	pH_4_END:
		IF timerDoCalibration.Q THEN
			timerDoCalibration.IN := FALSE;
			bBusy := FALSE;
			eSMState := WAIT;
		END_IF
	
	
	pH_10_START:
		nCalOutputPH10 := TRUE;
		timerBtnPress.IN := TRUE;
		IF timerBtnPress.Q THEN
			nCalOutputPH10 := FALSE;
			eSMState := pH_10_END;
			timerBtnPress.IN := FALSE; 
			timerDoCalibration.IN := TRUE;
		END_IF
		
		eSMState := pH_10_END;
			
			
		
	pH_10_END:
		IF timerDoCalibration.Q THEN
			timerDoCalibration.IN := FALSE;
			bBusy := FALSE;
			eSMState := WAIT;
		END_IF

END_CASE

METHOD PRIVATE calculate : BOOL
VAR_INPUT
	
	// Var
END_VAR
VAR
	nMeasuredCurrent: REAL;
END_VAR
nMeasuredCurrent := (INT_TO_REAL(nRawInput)/GVL.nMaxADCOutput)*16.0 + 4.0; // in mA

// nCurrentValue := (nMeasuredCurrent - 4.0) * (14.0 / 16.0);  // equation is PH = (mA reading - 4.0) * (14.0 / 16.0)
nCurrentValue := (nMeasuredCurrent - 4.0) * (14.0 / 16.0);  // equation is PH = (mA reading - 4.0) * (14.0 / 16.0)
END_METHOD

METHOD calibrate : BOOL
VAR_INPUT
	PhUnderTest: INT; // Can be 4, 7, or 10 (7 must be done first if doing multiple)
END_VAR
CASE PhUnderTest OF
	4:
		eSMState := pH_4_START;
	7:
		eSMState := pH_7_START;
	10:
		eSMState := pH_10_START;
END_CASE

bBusy := TRUE;
END_METHOD

{warning 'add method implementation '}
METHOD disable : BOOL
bEnable := FALSE;
END_METHOD

{warning 'add method implementation '}
METHOD enable : BOOL
bEnable := TRUE;
END_METHOD

{warning 'add method implementation '}
METHOD FB_init : BOOL
VAR_INPUT
	(* if TRUE, the retain variables are initialized (warm start / cold start)*)
	bInitRetains	: BOOL;
	(* if TRUE, the instance afterwards gets moved into the copy code (online change)*)
	bInCopyCode	: BOOL;
	
	SensorID	: STRING(80);
	SensorDescr	: STRING(255);
	SensorType	: E_SensorType;
END_VAR
sID := SensorID;
sDescr := SensorDescr;
eSensorType := SensorType;
END_METHOD

{warning 'add method implementation '}
METHOD getType : E_SensorType
getType := eSensorType;
END_METHOD

{warning 'add method implementation '}
METHOD getValue : REAL
getValue := nCurrentValue;
END_METHOD

{warning 'add method implementation '}
METHOD write : BOOL
// use this method to initiated a hardware read from assigned IO if required
END_METHOD

END_FUNCTION_BLOCK

// ---- POUs/02 Sensors/Dosing Machine/FB_Sensor_AtlasTEMP.TcPOU
{attribute 'OPC.UA.DA.StructuredType' := '1'}
FUNCTION_BLOCK FB_Sensor_AtlasTEMP EXTENDS FB_BaseDevice IMPLEMENTS I_Device, I_Sensor


VAR
	{attribute 'OPC.UA.DA' := '0'} 
	eSensorType: E_SensorType;
	{attribute 'OPC.UA.DA' := '0'} 
	nRawInput AT %I*: INT;
	nFaultInput AT %I*: BOOL;
	{attribute 'OPC.UA.DA' := '1'} 
	nCurrentValue: REAL;
	
	{attribute 'OPC.UA.DA' := '0'} 
	nCalOutput1 AT %Q*: BOOL;
	{attribute 'OPC.UA.DA' := '0'} 
	nCalOutput2 AT %Q*: BOOL;
	{attribute 'OPC.UA.DA' := '0'} 
	nCalOutput3 AT %Q*: BOOL;
	
	{attribute 'OPC.UA.DA' := '0'} 
	trigCalibrate: R_TRIG;
	{attribute 'OPC.UA.DA' := '0'} 
	timerBtnPress: TON := (PT:=T#250MS,IN := FALSE);
	
	{attribute 'OPC.UA.DA' := '0'} 
	timerDoCalibration: TON := (PT:=T#120S,IN := FALSE); // Check this time during testing! The instructions are not clear about what happens after initiating a calibration request 
	
	{attribute 'OPC.UA.DA' := '0'} 
	eSMState: (WAIT, CAL_START, CAL_FINISH) := WAIT;
	
END_VAR

calculate();

CASE eSMState OF 
	WAIT:
		// wait for the calibrate method call to change the ESMState variable
		
	CAL_START:
		nCalOutput1 := TRUE;
		timerBtnPress.IN := TRUE;
		IF timerBtnPress.Q THEN
			nCalOutput1 := FALSE;
			eSMState := CAL_FINISH;
			timerBtnPress.IN := FALSE; 
			timerDoCalibration.IN := TRUE;
		END_IF
		
		eSMState := CAL_FINISH;
		
	CAL_FINISH:
		IF timerDoCalibration.Q THEN
			timerDoCalibration.IN := FALSE;			// CHeck the functionality of this step - instructions are not clear
			bBusy := FALSE;
			eSMState := WAIT;
		END_IF
		
END_CASE

METHOD PRIVATE calculate : BOOL
VAR_INPUT
	
	// Var
END_VAR

VAR
	nMeasuredCurrent: REAL;
END_VAR
nMeasuredCurrent := (INT_TO_REAL(nRawInput)/GVL.nMaxADCOutput)*16.0 + 4.0; // in mA


nCurrentValue := (((nMeasuredCurrent - 4.0) / 16.0) * 360.0)- 180;  // equation is TEMP =    [(mA reading - 4.0)* 275 / 16 ] - 55

// nCurrentValue := (((nMeasuredCurrent - 4.0) * 275.0 / 16.0))- 55;  // equation is TEMP =    [(mA reading - 4.0)* 275 / 16 ] - 55

// This equation is for the default probe type 'Option 1' with a range of -55 to 220 deg C
END_METHOD

METHOD calibrate : BOOL
VAR_INPUT
END_VAR
// The user manual only shows a manual calibration method
// Perhaps this probe does not need to be calibrated as often and the PLC method is not offered? Need to investigate

eSMState := CAL_START;
END_METHOD

{warning 'add method implementation '}
METHOD disable : BOOL
bEnable := FALSE;
END_METHOD

{warning 'add method implementation '}
METHOD enable : BOOL
bEnable := TRUE;
END_METHOD

{warning 'add method implementation '}
METHOD FB_init : BOOL
VAR_INPUT
	(* if TRUE, the retain variables are initialized (warm start / cold start)*)
	bInitRetains	: BOOL;
	(* if TRUE, the instance afterwards gets moved into the copy code (online change)*)
	bInCopyCode	: BOOL;
	
	SensorID	: STRING(80);
	SensorDescr	: STRING(255);
	SensorType	: E_SensorType;
END_VAR
sID := SensorID;
sDescr := SensorDescr;
eSensorType := SensorType;
END_METHOD

{warning 'add method implementation '}
METHOD getType : E_SensorType
getType := eSensorType;
END_METHOD

{warning 'add method implementation '}
METHOD getValue : REAL
getValue := nCurrentValue;
END_METHOD

{warning 'add method implementation '}
METHOD write : BOOL
// use this method to initiated a hardware read from assigned IO if required
END_METHOD

END_FUNCTION_BLOCK

// ---- POUs/02 Sensors/Dosing Machine/FB_Sensor_GrowMedium_EC.TcPOU
{attribute 'OPC.UA.DA.StructuredType' := '1'}
FUNCTION_BLOCK FB_Sensor_GrowMedium_EC EXTENDS FB_BaseSensor IMPLEMENTS I_Device, I_Sensor

VAR
	
	bCAL: BOOL := FALSE;
	
	eSMState: (WAIT, CAL_LOW, CAL_HIGH, CALC_CORRECTION) := WAIT;

END_VAR
	
VAR PERSISTENT ;
	nECLOW_val: REAL;
	nECHIGH_val: REAL;
	
	nCurveGradient: REAL := 0.625; // 
	nCurveOffset: REAL := -2.5; // Defaults
END_VAR

calculate();
filter();

// Detect if any buttons in ignition have been pressed for Calibration
IF bCAL THEN 
	bCAL := FALSE;
	CASE eSMState OF
		WAIT:
			eSMState := CAL_LOW;
		CAL_LOW:
			eSMState := CAL_HIGH;
		CAL_HIGH:
			eSMState := CALC_CORRECTION;
	END_CASE
END_IF


CASE eSMState OF 
	WAIT:
		// wait here for a calibration command to be received
		eState := E_DeviceState.RUNNING;


	CAL_LOW:
		nECLOW_val := nMeasuredCurrent;
		eState := E_DeviceState.CAL_STEP1;

	CAL_HIGH:
		nECHIGH_val := nMeasuredCurrent;
		eState := E_DeviceState.CAL_STEP2;
	
	CALC_CORRECTION:
		nCurveGradient := ((1413.0-84.0)/1000.0) / (nECHIGH_val - nECLOW_val);
		nCurveOffset := (84.0/1000.0) - (nCurveGradient * nECLOW_val);
		eSMState := WAIT;
		eState := E_DeviceState.CAL_STEP3;
		
		
END_CASE

METHOD PRIVATE calculate : BOOL
VAR_INPUT
	
END_VAR
nMeasuredCurrent := (INT_TO_REAL(nRawInput)/GVL.nMaxADCOutput)*16.0 + 4.0; // in mA

// nCurrentValue := (nCurveGradient * nMeasuredCurrent) + nCurveOffset;

nCurrentValue := (nCurveGradient * nFilteredCurrent) + nCurveOffset; // delete this eventually
END_METHOD

METHOD calibrate : BOOL
VAR_INPUT
	
END_VAR
bCAL := TRUE;
END_METHOD

{warning 'add method implementation '}
METHOD disable : BOOL
bEnable := FALSE;
END_METHOD

{warning 'add method implementation '}
METHOD enable : BOOL
bEnable := TRUE;
END_METHOD

{warning 'add method implementation '}
METHOD FB_init : BOOL
VAR_INPUT
	(* if TRUE, the retain variables are initialized (warm start / cold start)*)
	bInitRetains	: BOOL;
	(* if TRUE, the instance afterwards gets moved into the copy code (online change)*)
	bInCopyCode	: BOOL;
	
	SensorID	: STRING(80);
	SensorDescr	: STRING(255);
	SensorType	: E_SensorType;
END_VAR
sID := SensorID;
sDescr := SensorDescr;
eSensorType := SensorType;
END_METHOD

{warning 'add method implementation '}
METHOD getType : E_SensorType
getType := eSensorType;
END_METHOD

{warning 'add method implementation '}
METHOD getValue : REAL
getValue := nCurrentValue;
END_METHOD

{warning 'add method implementation '}
METHOD write : BOOL
// use this method to initiated a hardware read from assigned IO if required
END_METHOD

END_FUNCTION_BLOCK

// ---- POUs/02 Sensors/Dosing Machine/FB_Sensor_GrowMedium_MOISTURE.TcPOU
{attribute 'OPC.UA.DA.StructuredType' := '1'}
FUNCTION_BLOCK FB_Sensor_GrowMedium_MOISTURE EXTENDS FB_BaseSensor IMPLEMENTS I_Device, I_Sensor

VAR
	
	bCAL: BOOL := FALSE;
	
	eSMState: (WAIT, CAL_DRY, CAL_WET, CALC_CORRECTION) := WAIT;

END_VAR
	
VAR PERSISTENT ;
	nMoisture_LOW_val: REAL;
	nMoisture_HIGH_val: REAL;
	
	nCurveGradient: REAL := 0.625; // 
	nCurveOffset: REAL := -2.5; // Defaults
END_VAR

calculate();
filter();

// Detect if any buttons in ignition have been pressed for Calibration
IF bCAL THEN 
	bCAL := FALSE;
	CASE eSMState OF
		WAIT:
			eSMState := CAL_DRY;
		CAL_DRY:
			eSMState := CAL_WET;
		CAL_WET:
			eSMState := CALC_CORRECTION;
	END_CASE
END_IF


CASE eSMState OF 
	WAIT:
		// wait here for a calibration command to be received
		eState := E_DeviceState.RUNNING;
	CAL_DRY:
		nMoisture_LOW_val 	:= nMeasuredCurrent;
		eState := E_DeviceState.CAL_STEP1;

	CAL_WET:
		nMoisture_HIGH_val 	:= nMeasuredCurrent;
		eState := E_DeviceState.CAL_STEP2;

	CALC_CORRECTION:
		nCurveGradient := 100.0 / (nMoisture_HIGH_val - nMoisture_LOW_val);
		nCurveOffset := 100.0 - (nCurveGradient * nMoisture_HIGH_val);
		eState := E_DeviceState.CAL_STEP3;
		eSMState := WAIT;
		
END_CASE

METHOD PRIVATE calculate : BOOL
VAR_INPUT
	
END_VAR
nMeasuredCurrent := (INT_TO_REAL(nRawInput)/GVL.nMaxADCOutput)*16.0 + 4.0; // in mA

// nCurrentValue := (nCurveGradient * nMeasuredCurrent) + nCurveOffset;

nCurrentValue := (nCurveGradient * nFilteredCurrent) + nCurveOffset; // delete this eventually
END_METHOD

METHOD calibrate : BOOL
VAR_INPUT
	
END_VAR

bCAL := TRUE;
END_METHOD

{warning 'add method implementation '}
METHOD disable : BOOL
bEnable := FALSE;
END_METHOD

{warning 'add method implementation '}
METHOD enable : BOOL
bEnable := TRUE;
END_METHOD

{warning 'add method implementation '}
METHOD FB_init : BOOL
VAR_INPUT
	(* if TRUE, the retain variables are initialized (warm start / cold start)*)
	bInitRetains	: BOOL;
	(* if TRUE, the instance afterwards gets moved into the copy code (online change)*)
	bInCopyCode	: BOOL;
	
	SensorID	: STRING(80);
	SensorDescr	: STRING(255);
	SensorType	: E_SensorType;
END_VAR
sID := SensorID;
sDescr := SensorDescr;
eSensorType := SensorType;
END_METHOD

{warning 'add method implementation '}
METHOD getType : E_SensorType
getType := eSensorType;
END_METHOD

{warning 'add method implementation '}
METHOD getValue : REAL
getValue := nCurrentValue;
END_METHOD

{warning 'add method implementation '}
METHOD write : BOOL
// use this method to initiated a hardware read from assigned IO if required
END_METHOD

END_FUNCTION_BLOCK

// ---- POUs/02 Sensors/Dosing Machine/FB_Sensor_GrowMedium_PH.TcPOU
{attribute 'OPC.UA.DA.StructuredType' := '1'}
FUNCTION_BLOCK FB_Sensor_GrowMedium_PH EXTENDS FB_BaseSensor IMPLEMENTS I_Device, I_Sensor

VAR

	bCAL: BOOL := FALSE;
	eSMState: (WAIT, CAL_4, CAL_7, CALC_CORRECTION) := WAIT;
	
END_VAR
	
VAR PERSISTENT 

	nPH4_val: REAL;
	nPH7_val: REAL;
	
	b4High_0_20High_1: BOOL := TRUE;
	
	nCurveGradient: REAL := 6.0/16.0; // Sensor range is PH 3 to 9 over 16mA range (4-20mA)
	nCurveOffset: REAL := 1.5; 
END_VAR

calculate();
filter();

// Detect if any buttons in ignition have been pressed for Calibration
IF bCAL THEN 
	bCAL := FALSE;
	CASE eSMState OF
		WAIT:
			eSMState := CAL_4;
		CAL_4:
			eSMState := CAL_7;
		CAL_7:
			eSMState := CALC_CORRECTION;
	END_CASE
END_IF




CASE eSMState OF 
	WAIT:
		// wait here for a calibration command to be received
		eState := E_DeviceState.RUNNING;
		
	CAL_4:
		nPH4_val := nFilteredCurrent;
		eState := E_DeviceState.CAL_STEP1;

	CAL_7:
		nPH7_val := nFilteredCurrent;
		eState := E_DeviceState.CAL_STEP2;

	CALC_CORRECTION:
		nCurveGradient := 3.0 / (nPH7_val - nPH4_val);
		nCurveOffset := 4.0 - (nCurveGradient * nPH4_val);
		eState := E_DeviceState.CAL_STEP3;
		eSMState := WAIT;
		
END_CASE

METHOD PRIVATE calculate : BOOL
VAR_INPUT
	
END_VAR
IF b4High_0_20High_1 THEN
	nMeasuredCurrent := (INT_TO_REAL(nRawInput)/GVL.nMaxADCOutput)*16.0 + 4.0; // in mA
ELSE
	nMeasuredCurrent := 20.0 - (INT_TO_REAL(nRawInput)/GVL.nMaxADCOutput)*16.00; 
END_IF


// nCurrentValue := (nCurveGradient * nMeasuredCurrent) + nCurveOffset; 

nCurrentValue := (nCurveGradient * nFilteredCurrent) + nCurveOffset; // delete this eventually

nCurrentValueFiltered := (nCurveGradient * nFilteredCurrent) + nCurveOffset;
END_METHOD

METHOD calibrate : BOOL
VAR_INPUT
	
END_VAR

bCAL := TRUE;
END_METHOD

{warning 'add method implementation '}
METHOD disable : BOOL
bEnable := FALSE;
END_METHOD

{warning 'add method implementation '}
METHOD enable : BOOL
bEnable := TRUE;
END_METHOD

{warning 'add method implementation '}
METHOD FB_init : BOOL
VAR_INPUT
	(* if TRUE, the retain variables are initialized (warm start / cold start)*)
	bInitRetains	: BOOL;
	(* if TRUE, the instance afterwards gets moved into the copy code (online change)*)
	bInCopyCode	: BOOL;
	
	SensorID	: STRING(80);
	SensorDescr	: STRING(255);
	SensorType	: E_SensorType;
END_VAR
sID := SensorID;
sDescr := SensorDescr;
eSensorType := SensorType;
END_METHOD

{warning 'add method implementation '}
METHOD getType : E_SensorType
getType := eSensorType;
END_METHOD

{warning 'add method implementation '}
METHOD getValue : REAL
getValue := nCurrentValue;
END_METHOD

{warning 'add method implementation '}
METHOD write : BOOL
// use this method to initiated a hardware read from assigned IO if required
END_METHOD

END_FUNCTION_BLOCK

// ---- POUs/02 Sensors/Dosing Machine/FB_Sensor_IFM_PG2453.TcPOU
{attribute 'OPC.UA.DA.StructuredType' := '1'}
FUNCTION_BLOCK FB_Sensor_IFM_PG2453 EXTENDS FB_BaseDevice IMPLEMENTS I_Device, I_Sensor

VAR

	{attribute 'OPC.UA.DA' := '0'} 
	eSensorType: E_SensorType;
	{attribute 'OPC.UA.DA' := '0'} 
	nRawInput AT %I*: INT;
	{attribute 'OPC.UA.DA' := '1'} 
	nCurrentValue: REAL;
	
	{attribute 'OPC.UA.DA' := '1'} 
	nVal4mA: REAL;
	{attribute 'OPC.UA.DA' := '1'} 
	nVal20mA: REAL;
END_VAR

calculate();

METHOD calculate : BOOL
VAR_INPUT
END_VAR
nCurrentValue := nVal4mA + (INT_TO_REAL(nRawInput) / GVL.nMaxADCOutput) * (nVal20mA - nVal4mA) ;
END_METHOD

{warning 'add method implementation '}
METHOD disable : BOOL
bEnable := FALSE;
END_METHOD

{warning 'add method implementation '}
METHOD enable : BOOL
bEnable := TRUE;
END_METHOD

{warning 'add method implementation '}
METHOD FB_init : BOOL
VAR_INPUT
	(* if TRUE, the retain variables are initialized (warm start / cold start)*)
	bInitRetains	: BOOL;
	(* if TRUE, the instance afterwards gets moved into the copy code (online change)*)
	bInCopyCode	: BOOL;
	SensorID	: STRING(80);
	SensorDescr	: STRING(255);
	SensorType	: E_SensorType;
	
END_VAR
sID := SensorID;
sDescr := SensorDescr;
eSensorType := SensorType;
END_METHOD

{warning 'add method implementation '}
METHOD getType : E_SensorType
getType := eSensorType;
END_METHOD

{warning 'add method implementation '}
METHOD getValue : REAL
getValue := nCurrentValue;
END_METHOD

METHOD setLimits : BOOL
VAR_INPUT
	Val_4mA: 	REAL;
	Val_20mA: 	REAL;
END_VAR
nVal4mA := Val_4mA;
nVal20mA := Val_20mA;
END_METHOD

{warning 'add method implementation '}
METHOD write : BOOL
END_METHOD

END_FUNCTION_BLOCK

// ---- POUs/02 Sensors/Dosing Machine/FB_Sensor_OceanControlsPressureTx_BVS006NA.TcPOU
{attribute 'OPC.UA.DA.StructuredType' := '1'}
FUNCTION_BLOCK FB_Sensor_OceanControlsPressureTx_BVS006NA EXTENDS FB_BaseDevice IMPLEMENTS I_Device, I_Sensor
// This is a 0 to 6BAR pressure sensor from 4mA to 20mA

VAR

	{attribute 'OPC.UA.DA' := '0'} 
	eSensorType: E_SensorType;
	{attribute 'OPC.UA.DA' := '0'} 
	nRawInput AT %I*: INT;
	{attribute 'OPC.UA.DA' := '1'} 
	nCurrentValue: REAL;
	
	{attribute 'OPC.UA.DA' := '1'} 
	nVal4mA: REAL := 0; //kPA
	{attribute 'OPC.UA.DA' := '1'} 
	nVal20mA: REAL := 600; //kPA
	
END_VAR

calculate();

METHOD calculate : BOOL
VAR_INPUT
END_VAR
nCurrentValue := nVal4mA + (INT_TO_REAL(nRawInput) / GVL.nMaxADCOutput) * (nVal20mA - nVal4mA) ;
END_METHOD

{warning 'add method implementation '}
METHOD disable : BOOL
bEnable := FALSE;
END_METHOD

{warning 'add method implementation '}
METHOD enable : BOOL
bEnable := TRUE;
END_METHOD

{warning 'add method implementation '}
METHOD FB_init : BOOL
VAR_INPUT
	(* if TRUE, the retain variables are initialized (warm start / cold start)*)
	bInitRetains	: BOOL;
	(* if TRUE, the instance afterwards gets moved into the copy code (online change)*)
	bInCopyCode	: BOOL;
	SensorID	: STRING(80);
	SensorDescr	: STRING(255);
	SensorType	: E_SensorType;
	
END_VAR
sID := SensorID;
sDescr := SensorDescr;
eSensorType := SensorType;
END_METHOD

{warning 'add method implementation '}
METHOD getType : E_SensorType
getType := eSensorType;
END_METHOD

{warning 'add method implementation '}
METHOD getValue : REAL
getValue := nCurrentValue;
END_METHOD

METHOD setLimits : BOOL
VAR_INPUT
	Val_4mA: 	REAL;
	Val_20mA: 	REAL;
END_VAR
nVal4mA := Val_4mA;
nVal20mA := Val_20mA;
END_METHOD

{warning 'add method implementation '}
METHOD write : BOOL
END_METHOD

END_FUNCTION_BLOCK

// ---- POUs/02 Sensors/Dosing Machine/FB_Sensor_SICKLevelSwitch_GRF18S.TcPOU
{attribute 'OPC.UA.DA.StructuredType' := '1'}
FUNCTION_BLOCK FB_Sensor_SICKLevelSwitch_GRF18S EXTENDS FB_BaseDevice IMPLEMENTS I_Device, I_Sensor

VAR
	
	{attribute 'OPC.UA.DA' := '0'} 
	eSensorType: E_SensorType;
	{attribute 'OPC.UA.DA' := '0'} 
	nRawInput AT %I*: BOOL;
	{attribute 'OPC.UA.DA' := '1'} 
	nCurrentValue: REAL;
END_VAR

calculate();

METHOD calculate : BOOL
VAR_INPUT
END_VAR
IF nRawInput THEN
	nCurrentValue := 1;
ELSE
	nCurrentValue := 0;
END_IF
END_METHOD

{warning 'add method implementation '}
METHOD disable : BOOL
bEnable := FALSE;
END_METHOD

{warning 'add method implementation '}
METHOD enable : BOOL
bEnable := TRUE;
END_METHOD

{warning 'add method implementation '}
METHOD FB_init : BOOL
VAR_INPUT
	(* if TRUE, the retain variables are initialized (warm start / cold start)*)
	bInitRetains	: BOOL;
	(* if TRUE, the instance afterwards gets moved into the copy code (online change)*)
	bInCopyCode	: BOOL;
	SensorID	: STRING(80);
	SensorDescr	: STRING(255);
	SensorType	: E_SensorType;
END_VAR
sID := SensorID;
sDescr := SensorDescr;
eSensorType := SensorType;
END_METHOD

{warning 'add method implementation '}
METHOD getType : E_SensorType
getType := eSensorType;
END_METHOD

{warning 'add method implementation '}
METHOD getValue : REAL
getValue := nCurrentValue;
END_METHOD

{warning 'add method implementation '}
METHOD write : BOOL
calculate();
END_METHOD

END_FUNCTION_BLOCK

// ---- POUs/02 Sensors/FB_DualRedundantSensor.TcPOU
{attribute 'OPC.UA.DA.StructuredType' := '1'}
FUNCTION_BLOCK FB_DualRedundantSensor EXTENDS FB_BaseDevice IMPLEMENTS I_Device, I_Sensor

VAR
	{attribute 'OPC.UA.DA' := '1'}
  	{attribute 'OPC.UA.DA.StructuredType' := '1'}
	fbSensor1: REFERENCE TO I_Sensor;
	{attribute 'OPC.UA.DA' := '1'}
  	{attribute 'OPC.UA.DA.StructuredType' := '1'}
	fbSensor2: REFERENCE TO I_Sensor;
	{attribute 'OPC.UA.DA' := '1'}
	nCurrentValue: REAL;
	
	eSensorType: E_SensorType;
	
	{attribute 'OPC.UA.DA' := '0'} 
	fbSenso1_vals: ARRAY[1..200] OF REAL;  //Arrays to store last 200 samples of sensors, enabling historic analysis
	{attribute 'OPC.UA.DA' := '0'} 
	fbSenso2_vals: ARRAY[1..200] OF REAL;
	
END_VAR

calculate();

METHOD addSensors : BOOL
VAR_INPUT
	
	Sensor1: REFERENCE TO I_Sensor;
	Sensor2: REFERENCE TO I_Sensor;
	
END_VAR

fbSensor1 := Sensor1;
fbSensor2 := Sensor2;
END_METHOD

METHOD calculate : BOOL
VAR_INPUT
END_VAR
//nCurrentValue := ( fbSensor1.getValue() + fbSensor2.getValue() ) / 2.0;  // calculate average of 2 sensors and return
END_METHOD

METHOD checkCorrelation : BOOL
VAR_INPUT
END_VAR
END_METHOD

{warning 'add method implementation '}
METHOD disable : BOOL
END_METHOD

{warning 'add method implementation '}
METHOD enable : BOOL
END_METHOD

{warning 'add method implementation '}
METHOD FB_init : BOOL
VAR_INPUT
	(* if TRUE, the retain variables are initialized (warm start / cold start)*)
	bInitRetains	: BOOL;
	(* if TRUE, the instance afterwards gets moved into the copy code (online change)*)
	bInCopyCode	: BOOL;
	SensorID	: STRING(80);
	SensorDescr	: STRING(255);
	SensorType	: E_SensorType;
	

	
END_VAR
sID := SensorID;
sDescr := SensorDescr;
eSensorType := SensorType;
END_METHOD

{warning 'add method implementation '}
METHOD getType : E_SensorType
END_METHOD

{warning 'add method implementation '}
METHOD getValue : REAL
END_METHOD

{warning 'add method implementation '}
METHOD write : BOOL
END_METHOD

END_FUNCTION_BLOCK

// ---- POUs/02 Sensors/FB_Sensor_4_20mA_Generic.TcPOU
{attribute 'OPC.UA.DA.StructuredType' := '1'}
FUNCTION_BLOCK FB_Sensor_4_20mA_Generic EXTENDS FB_BaseDevice IMPLEMENTS I_Device, I_Sensor

VAR
	{attribute 'OPC.UA.DA' := '1'} 
	eSensorType: E_SensorType;
	{attribute 'OPC.UA.DA' := '0'} 
	nRawInput AT %I*: INT;
	{attribute 'OPC.UA.DA' := '1'} 
	nCurrentValue: REAL;
	
	{attribute 'OPC.UA.DA' := '1'} 
	nVal4mA: REAL;
	{attribute 'OPC.UA.DA' := '1'} 
	nVal20mA: REAL;
END_VAR

calculate();

METHOD calculate : BOOL
VAR_INPUT
END_VAR
nCurrentValue := nVal4mA + (INT_TO_REAL(nRawInput) / GVL.nMaxADCOutput) * (nVal20mA - nVal4mA) ;
END_METHOD

{warning 'add method implementation '}
METHOD disable : BOOL
bEnable := FALSE;
END_METHOD

{warning 'add method implementation '}
METHOD enable : BOOL
bEnable := TRUE;
END_METHOD

{warning 'add method implementation '}
METHOD FB_init : BOOL
VAR_INPUT
	(* if TRUE, the retain variables are initialized (warm start / cold start)*)
	bInitRetains	: BOOL;
	(* if TRUE, the instance afterwards gets moved into the copy code (online change)*)
	bInCopyCode	: BOOL;
	SensorID	: STRING(80);
	SensorDescr	: STRING(255);
	SensorType	: E_SensorType;
	

END_VAR
sID := SensorID;
sDescr := SensorDescr;
eSensorType := SensorType;
END_METHOD

{warning 'add method implementation '}
METHOD getType : E_SensorType
getType := eSensorType;
END_METHOD

{warning 'add method implementation '}
METHOD getValue : REAL
getValue := nCurrentValue;
END_METHOD

METHOD setLimits : BOOL
VAR_INPUT
	Val_4mA: 	REAL;
	Val_20mA: 	REAL;
END_VAR
nVal4mA := Val_4mA;
nVal20mA := Val_20mA;
END_METHOD

{warning 'add method implementation '}
METHOD write : BOOL
END_METHOD

END_FUNCTION_BLOCK

// ---- POUs/02 Sensors/FB_Sensor_VaisalaGMW90.TcPOU

(*
	Handles communication and control of a Vaisala GMW90 environment sensor (Temp, Humidity, CO2)
*)
{attribute 'OPC.UA.DA.StructuredType' := '1'}
FUNCTION_BLOCK FB_Sensor_VaisalaGMW90 EXTENDS FB_BaseDevice
VAR_INPUT
	nModbusUnitID: UINT; // slave ID of the sensor
END_VAR
VAR_OUTPUT
	{attribute 'OPC.UA.DA' := '1'}
	rCO2 : REAL;
	{attribute 'OPC.UA.DA' := '1'}
	rTemperature : REAL;
	{attribute 'OPC.UA.DA' := '1'}
	rHumidity : REAL;
	nErrorCount : INT;
	nReadAttempts : INT;
	
END_VAR
VAR
	nSensorValues : ARRAY[1..10] OF WORD;
	nErrorCodes : ARRAY[1..10] OF WORD;
	
	nWordsToRead_values : UINT := 3; // ( CO2;  Temp;  Hum)
	nWordsToRead_errors : UINT := 2; // The GMW90 has 16 bits for error codes

	nAdrFirstReg_CO2 : WORD := 256; // THE GMW90 stores its int value for CO2 value in register 256
	nAdrFirstReg_Error : WORD := 513; // the GMW90 stores its error codes in 0513 register
	
	bRequestCompleted : BOOL; // is set to True by FB_Master when read is completed (or failed)
	
	bReadingError : BOOL; // we are currently reading the error register
	bTest : BOOL;
	tReadDelay : TON;
	bReadTrigger : BOOL;
	bReading : BOOL;
	tReadDelayTime : TIME := T#10S;
	trigError : R_TRIG;
	trigRead : R_TRIG;
END_VAR


VAR_IN_OUT
	fbModbus : FB_ModbusMaster;
END_VAR


// the function block just reads the modbus registers over and over.
// It takes turns between reading the values and reading the error codes

// 10 second cycle timer...
tReadDelay(IN := NOT bReadTrigger, PT := tReadDelayTime);
bReadTrigger := tReadDelay.Q AND NOT fbModbus.isBusy();
IF tReadDelay.Q THEN
	bReading := TRUE;
END_IF

IF bEnable AND bReadTrigger (*bReading*) THEN

	IF NOT bReadingError THEN
		
		// read CO2, Hum and Temp
		fbModbus.readRegs(ReadRegsVals := ADR(nSensorValues),
			SlaveAddress := nModbusUnitID,
			QtyWordsToRead := nWordsToRead_values,
			AdrFirstSlaveRegisterRead := nAdrFirstReg_CO2,
			bRequestCompleted := ADR(bRequestCompleted)
		);
		
	END_IF
	
	IF bReadingError THEN
		// read the error codes
		fbModbus.readRegs(ReadRegsVals := ADR(nErrorCodes),
			SlaveAddress := nModbusUnitID,
			QtyWordsToRead := nWordsToRead_errors,
			AdrFirstSlaveRegisterRead := nAdrFirstReg_Error,
			bRequestCompleted := ADR(bRequestCompleted)
		);
	END_IF
	
	IF bRequestCompleted THEN
		// the read has finished, so map the outputs
		IF NOT bReadingError THEN
			// map the sensor values
			rCO2 := nSensorValues[1]; 
			rHumidity :=  nSensorValues[2] / 100.00; 
			rTemperature := nSensorValues[3] / 100.00; 
		ELSE
			// map the errors
			
		END_IF
		
		// reset flags and start again
		bRequestCompleted := FALSE;
		bReadingError := FALSE;
		bReading := FALSE;
	END_IF
	
END_IF

// read count
trigRead(CLK := bReadTrigger);
IF trigRead.Q THEN
	nReadAttempts := nReadAttempts + 1;
END_IF

END_FUNCTION_BLOCK

// ---- POUs/02 Sensors/FB_Sensor_VaisalaGMW90_R2.TcPOU
(*
	Handles communication and control of a Vaisala GMW90 environment sensor (Temp, Humidity, CO2)
*)
{attribute 'OPC.UA.DA.StructuredType' := '1'}
FUNCTION_BLOCK FB_Sensor_VaisalaGMW90_R2 EXTENDS FB_BaseDevice

VAR_INPUT
	nModbusUnitID: UINT; // slave ID of the sensor
END_VAR

VAR_IN_OUT
	fbModbusManager : FB_ModbusManager;
	
END_VAR

VAR_OUTPUT
	{attribute 'OPC.UA.DA' := '1'}
	rCO2 : REAL;
	{attribute 'OPC.UA.DA' := '1'}
	rTemperature : REAL;
	{attribute 'OPC.UA.DA' := '1'}
	rHumidity : REAL;

END_VAR

VAR
	fbTON_DataRefresh: TON := (PT := T#10S, IN := FALSE);
	bFirstRun: BOOL := TRUE;
	bResetTtimer: BOOL := FALSE;
	bEnableComms: BOOL := FALSE;
	nWordsToRead_values : UINT := 1; // ( CO2;  Temp;  Hum)
	nWordsToRead_errors : UINT := 2; // The GMW90 has 16 bits for error codes
	
	nAdrFirstReg_CO2 : WORD := 256; // THE GMW90 stores its int value for CO2 value in register 256
	nAdrFirstReg_Hum : WORD := 257; // THE GMW90 stores its int value for CO2 value in register 256
	nAdrFirstReg_Temp : WORD := 258; // THE GMW90 stores its int value for CO2 value in register 256
	
	nAdrFirstReg_Error : WORD := 513; // the GMW90 stores its error codes in 0513 register
	
	stModRequest_ReadCO2: ST_Modbus_ReadRequest;
	stModRequest_ReadHum: ST_Modbus_ReadRequest;
	stModRequest_ReadTemp: ST_Modbus_ReadRequest;
	
	stModRequest_ReadError: ST_Modbus_ReadRequest;
	
END_VAR

IF bFirstRun THEN
	fbTON_DataRefresh(IN := TRUE);
	bFirstRun := FALSE;
	init_ModbusRequests();
END_IF

IF bResetTtimer THEN
	fbTON_DataRefresh(IN := TRUE);
	bResetTtimer := FALSE;
END_IF

(*
IF nModbusUnitID <> 0 THEN
	bEnableComms := TRUE;
END_IF
*)

fbTON_DataRefresh();

IF fbTON_DataRefresh.Q AND bEnableComms THEN
	fbModbusManager.addRequest_Read_Vaisala(ReadRequest := ADR(stModRequest_ReadCO2));
	fbModbusManager.addRequest_Read_Vaisala(ReadRequest := ADR(stModRequest_ReadHum));
	fbModbusManager.addRequest_Read_Vaisala(ReadRequest := ADR(stModRequest_ReadTemp));
	//fbModbusManager.addRequest_Read(ReadRequest := ADR(stModRequest_ReadError));
	
	//fbModbusManager.addRequest_Read_Vaisala(ReadRequest := ADR(stModRequest_ReadCO2));
	//fbModbusManager.addRequest_Read_Vaisala(ReadRequest := ADR(stModRequest_ReadCO2));
	rCO2 := 			stModRequest_ReadCO2.ReadRegsVals[1]; 
	rHumidity :=  		stModRequest_ReadHum.ReadRegsVals[1] / 100.00; 
	rTemperature := 	stModRequest_ReadTemp.ReadRegsVals[1] / 100.00; 
	
	fbTON_DataRefresh(IN := FALSE);
	bResetTtimer := TRUE;
END_IF

METHOD init_ModbusRequests : BOOL
VAR_INPUT
END_VAR
stModRequest_ReadCO2.SlaveAddress := nModbusUnitID;			
stModRequest_ReadCO2.AdrFirstSlaveRegisterRead := nAdrFirstReg_CO2;
stModRequest_ReadCO2.QtyWordsToRead := 1;				
stModRequest_ReadCO2.bRequestAccepted := FALSE;
stModRequest_ReadCO2.bRequestCompleted := FALSE;
stModRequest_ReadCO2.ReadRegsVals := GVL.ModbusEmptyBuffer;

stModRequest_ReadHum.SlaveAddress := nModbusUnitID;			
stModRequest_ReadHum.AdrFirstSlaveRegisterRead := nAdrFirstReg_Hum;
stModRequest_ReadHum.QtyWordsToRead := 1;				
stModRequest_ReadHum.bRequestAccepted := FALSE;
stModRequest_ReadHum.bRequestCompleted := FALSE;
stModRequest_ReadHum.ReadRegsVals := GVL.ModbusEmptyBuffer;

stModRequest_ReadTemp.SlaveAddress := nModbusUnitID;			
stModRequest_ReadTemp.AdrFirstSlaveRegisterRead := nAdrFirstReg_Temp;
stModRequest_ReadTemp.QtyWordsToRead := 1;				
stModRequest_ReadTemp.bRequestAccepted := FALSE;
stModRequest_ReadTemp.bRequestCompleted := FALSE;
stModRequest_ReadTemp.ReadRegsVals := GVL.ModbusEmptyBuffer;


stModRequest_ReadError.SlaveAddress := nModbusUnitID;			
stModRequest_ReadError.AdrFirstSlaveRegisterRead := nAdrFirstReg_Error;
stModRequest_ReadError.QtyWordsToRead := nWordsToRead_errors;			
stModRequest_ReadError.bRequestAccepted := FALSE;
stModRequest_ReadError.bRequestCompleted := FALSE;
stModRequest_ReadError.ReadRegsVals := GVL.ModbusEmptyBuffer;
END_METHOD

END_FUNCTION_BLOCK

// ---- POUs/02 Sensors/FB_Sensor_VaisalaGMW90_R2_1.TcPOU
(*
	Handles communication and control of a Vaisala GMW90 environment sensor (Temp, Humidity, CO2)
*)
{attribute 'OPC.UA.DA.StructuredType' := '1'}
FUNCTION_BLOCK FB_Sensor_VaisalaGMW90_R2_1 EXTENDS FB_BaseDevice

VAR_INPUT
	nModbusUnitID: UINT; // slave ID of the sensor
END_VAR

VAR_IN_OUT
	fbModbusManager : FB_ModbusManager;
	
END_VAR

VAR_OUTPUT
	{attribute 'OPC.UA.DA' := '1'}
	rCO2 : REAL;
	{attribute 'OPC.UA.DA' := '1'}
	rTemperature : REAL;
	{attribute 'OPC.UA.DA' := '1'}
	rHumidity : REAL;

END_VAR

VAR PERSISTENT 
	tDataRefresh: TIME := T#1m;
	tWaitForReadings: TIME := T#17S;
	tWaitForTurnOff: TIME := T#100MS;
	tMsgTimeout: TIME := T#2S;
	bEnableComms: BOOL := FALSE;
END_VAR

VAR
	
	
	bReading: BOOL := FALSE;
	bFirstRun: BOOL := TRUE;
	bResetTtimer: BOOL := FALSE;
	
	nWordsToRead_values : UINT := 1; // ( CO2;  Temp;  Hum)
	nWordsToRead_errors : UINT := 2; // The GMW90 has 16 bits for error codes
	
	nAdrFirstReg_CO2 : WORD := 256; // THE GMW90 stores its int value for CO2 value in register 256
	nAdrFirstReg_Hum : WORD := 257; // THE GMW90 stores its int value for CO2 value in register 256
	nAdrFirstReg_Temp : WORD := 258; // THE GMW90 stores its int value for CO2 value in register 256
	
	nAdrFirstReg_Error : WORD := 513; // the GMW90 stores its error codes in 0513 register
	
	stModRequest_ReadCO2: ST_Modbus_ReadRequest;
	stModRequest_ReadHum: ST_Modbus_ReadRequest;
	stModRequest_ReadTemp: ST_Modbus_ReadRequest;
	
	stModRequest_ReadError: ST_Modbus_ReadRequest;
	
	bVaisalaPowerCtr AT %Q*: BOOL;
	
	
	eSMState: (WAIT, ON, READ, TURN_OFF) := WAIT;
	
	fbTON_WaitForReadings: TON := (PT := tWaitForReadings, IN := FALSE);
	fbTON_WaitForTurnOff: TON := (PT := tWaitForReadings, IN := FALSE);
	fbTON_DataRefresh: TON := (PT := tDataRefresh, IN := FALSE);
	fbTON_MsgTimeout: TON := (PT := tMsgTimeout, IN := FALSE);
END_VAR

fbTON_WaitForTurnOff(PT := tWaitForTurnOff);
fbTON_WaitForReadings(PT := tWaitForReadings);
fbTON_DataRefresh(PT := tDataRefresh);
fbTON_MsgTimeout(PT := tMsgTimeout);

bVaisalaPowerCtr := TRUE;		// THis is a remnant of the power cycle workaround implemented in R7, keep this line here until we rewire room 7

IF bEnableComms THEN 
	IF bFirstRun THEN
		fbTON_DataRefresh(IN := TRUE);
		bFirstRun := FALSE;
		init_ModbusRequests();
	END_IF
	
	IF bResetTtimer THEN
		fbTON_DataRefresh(IN := TRUE);
		bResetTtimer := FALSE;
	END_IF
	
	(*
	IF nModbusUnitID <> 0 THEN
		bEnableComms := TRUE;
	END_IF
	*)
	
	CASE eSMState OF
		WAIT:
			fbTON_DataRefresh(IN := TRUE, PT := tDataRefresh);
			IF fbTON_DataRefresh.Q THEN
				eSMState := ON;
				fbTON_DataRefresh(IN := FALSE);
			END_IF
		
		ON:
			fbTON_WaitForReadings(PT := tWaitForReadings, IN := TRUE);
			//bVaisalaPowerCtr := TRUE;
			IF fbTON_WaitForReadings.Q THEN
				eSMState := READ;
			END_IF
			
		READ:
			IF fbTON_WaitForReadings.Q THEN
				fbTON_WaitForReadings(IN := FALSE);
				fbModbusManager.addRequest_Read_Vaisala(ReadRequest := ADR(stModRequest_ReadCO2));
				fbTON_MsgTimeout(IN := TRUE);
			END_IF
			
			IF stModRequest_ReadCO2.bRequestCompleted OR fbTON_MsgTimeout.Q THEN
				stModRequest_ReadCO2.bRequestCompleted := FALSE;
				fbTON_MsgTimeout( IN := FALSE);
				fbTON_WaitForTurnOff(IN := TRUE);
			END_IF
			
			IF fbTON_WaitForTurnOff.Q THEN
				//bVaisalaPowerCtr := FALSE;
				eSMState := WAIT;
				fbTON_WaitForTurnOff(IN := FALSE);
			END_IF
			
	END_CASE
	
	rCO2 := 			stModRequest_ReadCO2.ReadRegsVals[1]; 
	rHumidity :=  		stModRequest_ReadCO2.ReadRegsVals[2] / 100.00; 
	rTemperature := 	stModRequest_ReadCO2.ReadRegsVals[3] / 100.00; 
	
	
	(*
	
	IF fbTON_DataRefresh.Q AND bEnableComms THEN
		
		IF NOT fbTON_WaitForReadings.Q AND NOT bReading THEN
			fbTON_WaitForReadings(IN := TRUE);
			bVaisalaPowerCtr := TRUE;				// Turn the vaisala unit on
			bReading := TRUE;
		END_IF
			
		IF fbTON_WaitForReadings.Q THEN			// We have waited for the unit to power on, now we read
			fbModbusManager.addRequest_Read_Vaisala(ReadRequest := ADR(stModRequest_ReadCO2));
			fbTON_WaitForReadings(IN := FALSE);
		END_IF
		
		IF (stModRequest_ReadCO2.bRequestCompleted = TRUE) THEN // Request has finished, we turn power off after a set amount of time
			stModRequest_ReadCO2.bRequestCompleted := FALSE;
			fbTON_WaitForTurnOff(IN := TRUE);
		END_IF
		IF fbTON_WaitForTurnOff.Q THEN
			bVaisalaPowerCtr := FALSE;
			fbTON_WaitForTurnOff(IN := FALSE);
			fbTON_DataRefresh(IN := FALSE); 
			bResetTtimer := TRUE;
			fbTON_WaitForReadings(IN := FALSE);
			bReading := FALSE;
		END_IF
	END_IF
		
		
	
		//fbModbusManager.addRequest_Read(ReadRequest := ADR(stModRequest_ReadError));
		
		//fbModbusManager.addRequest_Read_Vaisala(ReadRequest := ADR(stModRequest_ReadCO2));
		//fbModbusManager.addRequest_Read_Vaisala(ReadRequest := ADR(stModRequest_ReadCO2));
		
		
	*)
END_IF

METHOD init_ModbusRequests : BOOL
VAR_INPUT
END_VAR
stModRequest_ReadCO2.SlaveAddress := nModbusUnitID;			
stModRequest_ReadCO2.AdrFirstSlaveRegisterRead := nAdrFirstReg_CO2;
stModRequest_ReadCO2.QtyWordsToRead := 3;				
stModRequest_ReadCO2.bRequestAccepted := FALSE;
stModRequest_ReadCO2.bRequestCompleted := FALSE;
stModRequest_ReadCO2.ReadRegsVals := GVL.ModbusEmptyBuffer;

(*
stModRequest_ReadHum.SlaveAddress := nModbusUnitID;			
stModRequest_ReadHum.AdrFirstSlaveRegisterRead := nAdrFirstReg_Hum;
stModRequest_ReadHum.QtyWordsToRead := 1;				
stModRequest_ReadHum.bRequestAccepted := FALSE;
stModRequest_ReadHum.bRequestCompleted := FALSE;
stModRequest_ReadHum.ReadRegsVals := GVL.ModbusEmptyBuffer;

stModRequest_ReadTemp.SlaveAddress := nModbusUnitID;			
stModRequest_ReadTemp.AdrFirstSlaveRegisterRead := nAdrFirstReg_Temp;
stModRequest_ReadTemp.QtyWordsToRead := 1;				
stModRequest_ReadTemp.bRequestAccepted := FALSE;
stModRequest_ReadTemp.bRequestCompleted := FALSE;
stModRequest_ReadTemp.ReadRegsVals := GVL.ModbusEmptyBuffer;
*)

stModRequest_ReadError.SlaveAddress := nModbusUnitID;			
stModRequest_ReadError.AdrFirstSlaveRegisterRead := nAdrFirstReg_Error;
stModRequest_ReadError.QtyWordsToRead := nWordsToRead_errors;			
stModRequest_ReadError.bRequestAccepted := FALSE;
stModRequest_ReadError.bRequestCompleted := FALSE;
stModRequest_ReadError.ReadRegsVals := GVL.ModbusEmptyBuffer;
END_METHOD

END_FUNCTION_BLOCK

// ---- POUs/03 Physical Entities/FB_BagFilter.TcPOU
{attribute 'OPC.UA.DA.StructuredType' := '1'}
FUNCTION_BLOCK FB_BagFilter EXTENDS FB_BaseDevice IMPLEMENTS I_Device

VAR
	{attribute 'OPC.UA.DA' := '1'}
  	{attribute 'OPC.UA.DA.StructuredType' := '1'}
	fbDiffPress_Upstream: I_Sensor(SensorID := '', SensorDescr := '', SensorType := E_SensorType.Analogue);
	{attribute 'OPC.UA.DA' := '1'}
  	{attribute 'OPC.UA.DA.StructuredType' := '1'}
	fbDiffPress_Downstream: I_Sensor(SensorID := '', SensorDescr := '', SensorType := E_SensorType.Analogue);
	{attribute 'OPC.UA.DA' := '1'}
	nDiffPressure: REAL;
	
END_VAR

VAR_IN_OUT
	{attribute 'OPC.UA.DA' := '1'}
	nMaxPressure: UINT;
END_VAR

// Bag Filters do not actually do anything, however it will be useful to maintain an OEE object for these
// We can then monitor when filters need to be replaced

nDiffPressure := ABS(fbDiffPress_Upstream.getValue() - fbDiffPress_Downstream.getValue());

{warning 'add method implementation '}
METHOD disable : BOOL
END_METHOD

{warning 'add method implementation '}
METHOD enable : BOOL
END_METHOD

METHOD FB_init : BOOL
VAR_INPUT
	bInitRetains : BOOL; // if TRUE, the retain variables are initialized (warm start / cold start)
	bInCopyCode : BOOL;  // if TRUE, the instance afterwards gets moved into the copy code (online change)
	
	FilterID: STRING(80);
	FilterDescr: STRING(255);

END_VAR
sID := FilterID;
sDescr := FilterDescr;
END_METHOD

METHOD getDiffPressure : REAL
VAR_INPUT
END_VAR
//getDiffPressure := fbSensorPIT_Upstream.getValue() - fbSensorPIT_Downstream.getValue();
END_METHOD

METHOD setPressureLimits : BOOL
VAR_INPUT
	PressTx_Upstream: I_Sensor(SensorID := '', SensorDescr := '', SensorType := E_SensorType.Analogue);
	PressTx_Downstream: I_Sensor(SensorID := '', SensorDescr := '', SensorType := E_SensorType.Analogue);
END_VAR

fbDiffPress_Downstream := PressTx_Downstream;
fbDiffPress_Upstream := PressTx_Upstream;
END_METHOD

END_FUNCTION_BLOCK

// ---- POUs/03 Physical Entities/FB_Tank.TcPOU
{attribute 'OPC.UA.DA.StructuredType' := '1'}
FUNCTION_BLOCK FB_Tank EXTENDS FB_BaseDevice IMPLEMENTS I_Device

VAR
	{attribute 'OPC.UA.DA' := '1'}
	nFillSetPoint: REAL	;
	{attribute 'OPC.UA.DA' := '1'}
	nFillActual:   REAL;
	{attribute 'OPC.UA.DA' := '1'}
  	{attribute 'OPC.UA.DA.StructuredType' := '1'}	
	bSensorLL: BOOL := FALSE;
	{attribute 'OPC.UA.DA' := '1'}
  	{attribute 'OPC.UA.DA.StructuredType' := '1'}
	bSensorL: BOOL := FALSE;
	{attribute 'OPC.UA.DA' := '1'}
  	{attribute 'OPC.UA.DA.StructuredType' := '1'}
	bSensorH: BOOL := FALSE;
	{attribute 'OPC.UA.DA' := '1'}
  	{attribute 'OPC.UA.DA.StructuredType' := '1'}
	bSensorHH: BOOL := FALSE;
	{attribute 'OPC.UA.DA' := '1'}
  	{attribute 'OPC.UA.DA.StructuredType' := '1'}
	nSensorLIT: REAL := 0.0;
END_VAR
VAR_INPUT
	fbSensor_LL: I_Sensor(SensorID := '', SensorDescr := '' , 	SensorType := E_SensorType.Digital);
	fbSensor_L: I_Sensor(SensorID := '', SensorDescr := '' , 	SensorType := E_SensorType.Digital);
	fbSensor_H: I_Sensor(SensorID := '', SensorDescr := '' , 	SensorType := E_SensorType.Digital);
	fbSensor_HH: I_Sensor(SensorID := '', SensorDescr := '' , 	SensorType := E_SensorType.Digital);
	fbSensor_LIT: I_Sensor(SensorID := '', SensorDescr := '' , 	SensorType := E_SensorType.Analogue);
	
	bSensorLL_Enable: BOOL;
	bSensorL_Enable: BOOL;
	bSensorH_Enable: BOOL;
	bSensorHH_Enable: BOOL;
	bSensorLIT_Enable: BOOL;
END_VAR

update();

{warning 'add method implementation '}
METHOD disable : BOOL
END_METHOD

{warning 'add method implementation '}
METHOD enable : BOOL
END_METHOD

{warning 'add method implementation '}
METHOD FB_init : BOOL
VAR_INPUT
	(* if TRUE, the retain variables are initialized (warm start / cold start)*)
	bInitRetains	: BOOL;
	(* if TRUE, the instance afterwards gets moved into the copy code (online change)*)
	bInCopyCode	: BOOL;
	TankID	: STRING(80);
	TankDescr	: STRING(255);
	
END_VAR
sID := TankID;
sDescr := TankDescr;
END_METHOD

METHOD PRIVATE update : BOOL
VAR_INPUT
END_VAR

IF bSensorLL_Enable THEN
	IF fbSensor_LL.getValue() = 1 THEN
		bSensorLL := TRUE;
	ELSE
		bSensorLL := FALSE;
	END_IF
END_IF


IF bSensorL_Enable THEN
	IF fbSensor_L.getValue() = 1 THEN
		bSensorL := TRUE;
	ELSE
		bSensorL := FALSE;
	END_IF
END_IF

IF bSensorH_Enable THEN
	IF fbSensor_H.getValue() = 1 THEN
		bSensorH := TRUE;
	ELSE
		bSensorH := FALSE;
	END_IF
END_IF

IF bSensorHH_Enable THEN
	IF fbSensor_HH.getValue() = 1 THEN
		bSensorHH := TRUE;
	ELSE
		bSensorHH := FALSE;
	END_IF
END_IF

IF bSensorLIT_Enable THEN
	nSensorLIT := fbSensor_LIT.getValue();
END_IF
END_METHOD

END_FUNCTION_BLOCK

// ---- POUs/04 Control Loops/Dosing Machine/FB_BangBangControl.TcPOU

(*
	Function Block which performs a bang-bang control loop.
*)
{attribute 'OPC.UA.DA.StructuredType' := '1'}
FUNCTION_BLOCK FB_BangBangControl EXTENDS FB_BaseDevice
VAR_INPUT
	{attribute 'OPC.UA.DA' := '1'}
	rAlarmHigh : REAL;
	{attribute 'OPC.UA.DA' := '1'}
	rAlarmLow : REAL;
	{attribute 'OPC.UA.DA' := '1'}
	rLimitHigh : REAL; // the upper limit of the desirable range (when the downward adjustment is activated)
	{attribute 'OPC.UA.DA' := '1'}
	rLimitLow : REAL; // lower limit of the desirable range (when the upward adjustment is activated)
	{attribute 'OPC.UA.DA' := '1'}
	nAdjustDelay : REAL; // min time in seconds between adjustments
	{attribute 'OPC.UA.DA' := '1'}
	nAdjustDownDuration : REAL; // time in seconds that the downward adjustment output is turned on when performing a downward adjustment
	{attribute 'OPC.UA.DA' := '1'}
	nAdjustUpDuration : REAL; // time in seconds that the upward adjustment output is turned on when performing a upward adjustment
	{attribute 'OPC.UA.DA' := '1'}
	rCurrentValue : REAL; 
	{attribute 'OPC.UA.DA' := '1'}
	bEnabled : BOOL; 
	{attribute 'OPC.UA.DA' := '1'}
	sParameterName : STRING;
	{attribute 'OPC.UA.DA' := '1'}
	rSetpoint: REAL;
	{attribute 'OPC.UA.DA' := '1'}
	Mode:    E_CTRL_MODE;
END_VAR
VAR_OUTPUT
	{attribute 'OPC.UA.DA' := '1'}
	bAdjustDownOutput AT %Q*: BOOL;
	{attribute 'OPC.UA.DA' := '1'}
	bAdjustUpOutput AT %Q*: BOOL;
	{attribute 'OPC.UA.DA' := '1'}
	bAlarmHigh : BOOL;
	{attribute 'OPC.UA.DA' := '1'}
	bAlarmLow : BOOL;
END_VAR
VAR
	tAdjustDownTimer : TON;
	tAdjustUpTimer : TON;
	tAdjustDelayTimer : TON;
	bAdjustDownActive : BOOL;
	bAdjustUpActive : BOOL;
	bDelayActive : BOOL;
	
	//rProportionalGainUp: REAL := 0.0001;
	//rProportionalGainDown: REAL := 0.0001;
END_VAR



IF eState = E_DeviceState.RUNNING THEN
	timers();
	// output signals
	bAdjustDownOutput := bAdjustDownActive;
	bAdjustUpOutput := bAdjustUpActive;
	// alarms
	bAlarmHigh := (rCurrentValue >= rAlarmHigh);
	bAlarmLow := (rCurrentValue <= rAlarmLow);
ELSE
	bAdjustDownOutput := FALSE;
	bAdjustUpOutput := FALSE;
	bAlarmHigh := FALSE;
	bAlarmLow := FALSE;
	// clear the delay timer 
	tAdjustDelayTimer.PT := INT_TO_TIME(0);
END_IF

// update setpoint (just for historizing purposes)
rSetpoint := (rLimitHigh + rLimitLow) / 2.0;

METHOD setState : BOOL
VAR_INPUT
	state : E_DeviceState;
END_VAR

eState := state;
END_METHOD

(*
	Run the timers for delay, adjust up and adjust down
*)
METHOD timers : BOOL
VAR_INPUT
END_VAR

tAdjustDelayTimer(IN := bDelayActive, PT := REAL_TO_TIME(nAdjustDelay) * 1000);
tAdjustDownTimer(IN := bAdjustDownActive, PT := REAL_TO_TIME(nAdjustDownDuration) * 1000);
tAdjustUpTimer(IN := bAdjustUpActive, PT := REAL_TO_TIME(nAdjustUpDuration) * 1000);

IF tAdjustDelayTimer.Q THEN
	// the delay timer is finished so check if we need to activate an adjustment
	
	//bAdjustDownActive := rCurrentValue > ((rLimitHigh + rLimitLow) / 2.0)*1.025;
	bAdjustDownActive := rCurrentValue > (1.1 * rLimitHigh); // only exhaust if we are way over 
	bAdjustUpActive := rCurrentValue < ((rLimitHigh + rLimitLow) / 2.0)*0.985;
	
	//nAdjustUpDuration := (ABS(rCurrentValue - ((rLimitHigh + rLimitLow) / 2.0)) * rProportionalGainDown);
	//nAdjustDownDuration  := (ABS(rCurrentValue - ((rLimitHigh + rLimitLow) / 2.0)) * rProportionalGainUp);
END_IF

// run the delay timer whenever we are not activating an output
bDelayActive := NOT bAdjustDownActive AND NOT bAdjustUpActive;

// unlatch adjustDownActive when timer finishes
IF tAdjustDownTimer.Q THEN
	bAdjustDownActive := FALSE;
END_IF

// unlatch adjustUpActive when timer finishes
IF tAdjustUpTimer.Q THEN
	bAdjustUpActive := FALSE;
END_IF
END_METHOD

END_FUNCTION_BLOCK

// ---- POUs/04 Control Loops/Dosing Machine/FB_BangBangControl_Analog.TcPOU
(*
	Function Block which performs a bang-bang control loop.
*)
{attribute 'OPC.UA.DA.StructuredType' := '1'}
FUNCTION_BLOCK FB_BangBangControl_Analog EXTENDS FB_BaseDevice
VAR_INPUT PERSISTENT
	{attribute 'OPC.UA.DA' := '1'}
	rAlarmHigh : REAL;
	{attribute 'OPC.UA.DA' := '1'}
	rAlarmLow : REAL;
	{attribute 'OPC.UA.DA' := '1'}
	rLimitHigh : REAL; // the upper limit of the desirable range (when the downward adjustment is activated)
	{attribute 'OPC.UA.DA' := '1'}
	rLimitLow : REAL; // lower limit of the desirable range (when the upward adjustment is activated)
	{attribute 'OPC.UA.DA' := '1'}
	nAdjustDelay : INT := 30; // min time in seconds between adjustments
	{attribute 'OPC.UA.DA' := '1'}
	nAdjustDownIncrement : REAL := 0.5;
	{attribute 'OPC.UA.DA' := '1'}
	nAdjustUpIncrement : REAL := 0.5; 
	{attribute 'OPC.UA.DA' := '1'}
	rCurrentValue : REAL; 
	{attribute 'OPC.UA.DA' := '1'}
	bEnabled : BOOL; 
	{attribute 'OPC.UA.DA' := '1'}
	sParameterName : STRING;
	
	{attribute 'OPC.UA.DA' := '1'}
	nControlValue: POINTER TO REAL;
	{attribute 'OPC.UA.DA' := '1'}
	nControlValueCopy: REAL;
	
	{attribute 'OPC.UA.DA' := '1'}
	Mode:    E_CTRL_MODE;
END_VAR

VAR_OUTPUT

	{attribute 'OPC.UA.DA' := '1'}
	bAlarmHigh : BOOL;
	{attribute 'OPC.UA.DA' := '1'}
	bAlarmLow : BOOL;
END_VAR

VAR
	tAdjustDownTimer : TON;
	tAdjustUpTimer : TON;
	tAdjustDelayTimer : TON;
	bAdjustDownActive : BOOL;
	bAdjustUpActive : BOOL;
	bDelayActive : BOOL;
END_VAR

IF eState = E_DeviceState.RUNNING THEN
	timers();
	// output signals
	IF bAdjustUpActive THEN
		IF NOT (nControlValue^ > ((rLimitHigh + rLimitLow)/2.0)) THEN
			nControlValue^ := nControlValue^ + nAdjustUpIncrement;
		END_IF
		bAdjustUpActive := FALSE;	
	END_IF
	
	IF bAdjustDownActive THEN
		IF NOT (nControlValue^ <= 16) THEN
			nControlValue^ := nControlValue^ - nAdjustDownIncrement;
		END_IF
		bAdjustDownActive := FALSE;	
	END_IF
	
	// alarms
	bAlarmHigh := (rCurrentValue >= rAlarmHigh);
	bAlarmLow := (rCurrentValue <= rAlarmLow);
ELSE
	bAlarmHigh := FALSE;
	bAlarmLow := FALSE;
	// clear the delay timer 
	tAdjustDelayTimer.PT := INT_TO_TIME(0);
END_IF

nControlValueCopy := nControlValue^;

METHOD setState : BOOL
VAR_INPUT
	state : E_DeviceState;
END_VAR

eState := state;
END_METHOD


(*
	Run the timers for delay, adjust up and adjust down
*)
METHOD timers : BOOL
VAR_INPUT
END_VAR
tAdjustDelayTimer(IN := bDelayActive, PT := INT_TO_TIME(nAdjustDelay) * 1000);


IF tAdjustDelayTimer.Q THEN
	// the delay timer is finished so check if we need to activate an adjustment
	
	//bAdjustDownActive := (rCurrentValue > rLimitHigh);
	//bAdjustUpActive := (rCurrentValue < rLimitLow);
	
	bAdjustDownActive := (rCurrentValue > ((rLimitHigh + rLimitLow)/2.0)+0.6);
	bAdjustUpActive := (rCurrentValue < ((rLimitHigh + rLimitLow)/2.0)-0.6);
	
END_IF

// run the delay timer whenever we are not activating an output
bDelayActive := NOT bAdjustDownActive AND NOT bAdjustUpActive;
END_METHOD

END_FUNCTION_BLOCK

// ---- POUs/04 Control Loops/Dosing Machine/FB_BatchController_Dosing.TcPOU
FUNCTION_BLOCK FB_BatchController_Dosing EXTENDS FB_BaseDevice

VAR PERSISTENT
	nVolumeWater: REAL := 200.0; // Litres
	
	{attribute 'OPC.UA.DA' := '0'} 
	eCurrentNutrient: 			(NUTRIENT_A,NUTRIENT_B,NUTRIENT_C, PH) := NUTRIENT_C;
	
	benableDosPumps: BOOL := TRUE;
	
	{attribute 'OPC.UA.DA' := '1'} 
	nDoseQTY_Nutrient: 	INT;
	{attribute 'OPC.UA.DA' := '1'} 
	nDoseQTY_pH: 		INT;
	
	{attribute 'OPC.UA.DA' := '1'} 
	tPIDLoopTime: TIME := T#1M;	//5 second PID calculation

END_VAR

VAR
	bFirstRun: BOOL := TRUE;
	bResetTimer: BOOL := FALSE;
	
	{attribute 'OPC.UA.DA' := '0'} 
	fbSensor_EC:	I_Sensor(SensorID := '', SensorDescr := '' , SensorType := E_SensorType.Analogue);
	{attribute 'OPC.UA.DA' := '0'} 
	fbSensor_DO:	I_Sensor(SensorID := '', SensorDescr := '' , SensorType := E_SensorType.Analogue);
	{attribute 'OPC.UA.DA' := '0'} 
	fbSensor_ORP:	I_Sensor(SensorID := '', SensorDescr := '' , SensorType := E_SensorType.Analogue);
	{attribute 'OPC.UA.DA' := '0'} 
	fbSensor_PH:	I_Sensor(SensorID := '', SensorDescr := '' , SensorType := E_SensorType.Analogue);
	{attribute 'OPC.UA.DA' := '0'} 
	fbSensor_TEMP:	I_Sensor(SensorID := '', SensorDescr := '' , SensorType := E_SensorType.Analogue);	

	{attribute 'OPC.UA.DA' := '0'} 
	fbDosingPump_phUp:  		I_PumpDosing;
	{attribute 'OPC.UA.DA' := '0'} 
	fbDosingPump_phDOwn:  		I_PumpDosing;
	{attribute 'OPC.UA.DA' := '0'} 
	fbDosingPump_Nutrient_A:  	I_PumpDosing;
	{attribute 'OPC.UA.DA' := '0'} 
	fbDosingPump_Nutrient_B:  	I_PumpDosing;
	{attribute 'OPC.UA.DA' := '0'} 
	fbDosingPump_Nutrient_C:  	I_PumpDosing;
	{attribute 'OPC.UA.DA' := '0'} 
	eSMState: 					(WAIT, CALCULATE, NUTRIENT_ONLY, NUTRIENT_AND_PH, PH_ONLY) := WAIT;
	
END_VAR

METHOD calcError : BOOL
VAR_INPUT
END_VAR
nPIDNutrientError 	:= nPIDNutrientSetpoint - nNutrient_ProcessValue;
nPIDNutrientError 	:= nPIDNutrientError;

nPIDPHError			:= nPIDPHSetpoint_Moles - nPH_ProcessValue_Moles;
END_METHOD

METHOD calcInput : BOOL
VAR_INPUT
END_VAR
//nPIDPHSetpoint 			:= 	EXPT(10, -1.0 * fbSensor_PH.getValue());

nNutrient_ProcessValue 		:= 	fbSensor_EC.getValue();

//nPIDPHSetpoint 			:= 	EXPT(10, -1.0 * fbSensor_PH.getValue());

nPIDPHSetpoint_Moles		:= 	EXPT(10, -1.0 * nPH_Setpoint) * nVolumeWater;
nPH_ProcessValue_Moles		:= 	EXPT(10, -1.0 * fbSensor_PH.getValue())  * nVolumeWater;

nPH_ProcessValue			:= fbSensor_PH.getValue();
//nPH_Setpoint				:= fbSensor_PH.getValue();
nPH_HighBand				:= nPH_Setpoint + 0.1;
nPH_LowBand					:= nPH_Setpoint - 0.1;
END_METHOD

METHOD FB_init : BOOL
VAR_INPUT
	bInitRetains : BOOL; // if TRUE, the retain variables are initialized (warm start / cold start)
	bInCopyCode : BOOL;  // if TRUE, the instance afterwards gets moved into the copy code (online change)
	
	DosingPump_phUp:  			I_PumpDosing;
	DosingPump_phDOwn:  		I_PumpDosing;
	DosingPump_Nutrient_A:  	I_PumpDosing;
	DosingPump_Nutrient_B:  	I_PumpDosing;
	DosingPump_Nutrient_C:  	I_PumpDosing;
	
	Sensor_EC:				I_Sensor(SensorID := '', SensorDescr := '' , SensorType := E_SensorType.Analogue);
	Sensor_DO:				I_Sensor(SensorID := '', SensorDescr := '' , SensorType := E_SensorType.Analogue);
	Sensor_ORP:				I_Sensor(SensorID := '', SensorDescr := '' , SensorType := E_SensorType.Analogue);
	Sensor_PH:				I_Sensor(SensorID := '', SensorDescr := '' , SensorType := E_SensorType.Analogue);
	Sensor_TEMP:			I_Sensor(SensorID := '', SensorDescr := '' , SensorType := E_SensorType.Analogue);
	
END_VAR
fbDosingPump_phUp := DosingPump_phUp;
fbDosingPump_phDOwn := DosingPump_phDOwn;
fbDosingPump_Nutrient_A := DosingPump_Nutrient_A;
fbDosingPump_Nutrient_B := DosingPump_Nutrient_B;
fbDosingPump_Nutrient_C := DosingPump_Nutrient_C;

fbSensor_EC := Sensor_EC;
fbSensor_DO := Sensor_DO;
fbSensor_ORP := Sensor_ORP;
fbSensor_PH := Sensor_PH;
fbSensor_TEMP := Sensor_TEMP;
END_METHOD

METHOD setParams : BOOL
VAR_INPUT
	(*
	NutrientMaxDoseRate: UINT;
	NutrientMinDoseRate: UINT;
	NutrientTimeBetweenDoses: TIME;
	PHMaxDoseRate: UINT;
	PHMinDoseRate: UINT;
	PHTimeBetweenDoses: TIME;


	// PID loop variables below
	*)
	NutrientSetpoint:		REAL; 
	(*
	NutrientSetpointBand:	REAL;
	
	NutrientManSyncVal:		REAL;
	NutrientSync: 			BOOL; 
	NutrientHold: 			BOOL;
	NutrientMode: 			E_CTRL_MODE;
	NutrientCtrlCycleTime: 	TIME;
	NutrientTaskCycleTime:	TIME;
	
	//stPIDParams values
	NutrientKp:  				REAL;
	NutrientTn: 				TIME; 
	NutrientTv:					TIME; 
	NutrientTd:					TIME; 
	NutrientOutMaxLimit: 		REAL;
	NutrientOutMinLimit:		REAL;
	NutrientPInTheFeedbackPath: BOOL;
	NutrientDInTheFeedbackPath: BOOL;
	NutrientARWOnIPartOnly:		BOOL;
	
	*)
	PHSetpoint:			REAL; 
	PHSetpointBand:		REAL;
	(*
	PHManSyncVal:		REAL;
	PHSync: 			BOOL;
	PHHold: 			BOOL;
	PHMode: 			E_CTRL_MODE;
	PHCtrlCycleTime: 		TIME;
	PHTaskCycleTime:		TIME;
	
	
	//stPIDParams values
	*)
	PHKp:  					REAL;
	PHTn: 					TIME;
	PHTv:					TIME;
	PHTd:					TIME; 
	(*
	PHOutMaxLimit: 			REAL; 		
	PHOutMinLimit:			REAL;
	PHPInTheFeedbackPath: 	BOOL;
	PHDInTheFeedbackPath:	BOOL;
	PHARWOnIPartOnly:		BOOL;
	*)
	
END_VAR
(*
nPIDNutrientMaxDoseRate := 				NutrientMaxDoseRate;
nPIDNutrientMinDoseRate := 				NutrientMinDoseRate;
tPIDNutrientTimeBetweenDoses := 		NutrientTimeBetweenDoses;

nPIDPHMaxDoseRate := 					PHMaxDoseRate;
nPIDPHMinDoseRate := 					PHMinDoseRate;
tPIDPHTimeBetweenDoses := 				PHTimeBetweenDoses;

*)
nPIDNutrientSetpoint := 				NutrientSetpoint;
(*
nPIDNutrientSetpointBand := 			NutrientSetpointBand;
nPIDNutrientManSyncVal := 				NutrientManSyncVal;
bPIDNutrientSync := 					NutrientSync;
bPIDNutrientHold := 					NutrientHold;
ePIDNutrientMode := 					NutrientMode;
tPIDNutrientCtrlCycleTime := 			NutrientCtrlCycleTime;
tPIDNutrientTaskCycleTime := 			NutrientTaskCycleTime;

nPIDNutrientKp := 						NutrientKp;
tPIDNutrientTn := 						NutrientTn;
tPIDNutrientTv := 						NutrientTv;
tPIDNutrientTd := 						NutrientTd;
nPIDNutrientOutMaxLimit := 				NutrientOutMaxLimit;
nPIDNutrientOutMinLimit := 				NutrientOutMinLimit;
bPIDNutrientPInTheFeedbackPath := 		NutrientPInTheFeedbackPath;
bPIDNutrientDInTheFeedbackPath := 		NutrientDInTheFeedbackPath;
bPIDNutrientARWactive := 				NutrientARWOnIPartOnly;
*)
nPH_Setpoint := 						PHSetpoint;

nPIDPHSetpointBand := 					PHSetpointBand;
(*
nPIDPHManSyncVal := 					PHManSyncVal;
bPIDPHSync := 							PHSync;
bPIDPHHold := 							PHHold;
ePIDPHMode := 							PHMode;
tPIDPHCtrlCycleTime := 					PHCtrlCycleTime;
tPIDPHTaskCycleTime := 					PHTaskCycleTime;
*)
nPIDPHKp := 							PHKp;
tPIDPHTn := 							PHTn * 1000;
tPIDPHTv := 							PHTv * 1000;
tPIDPHTd := 							PHTd * 1000;
(*
nPIDPHOutMaxLimit := 					PHOutMaxLimit;
nPIDPHOutMinLimit := 					PHOutMinLimit;
bPIDPHPInTheFeedbackPath := 			PHPInTheFeedbackPath;
bPIDPHDInTheFeedbackPath := 			PHDInTheFeedbackPath;
bPIDPHARWactive := 						PHARWOnIPartOnly;
*)
END_METHOD

METHOD updatePIDParams : BOOL
VAR_INPUT
END_VAR
stPIDNutrientParameters.tCtrlCycleTime := tPIDNutrientCtrlCycleTime;
stPIDNutrientParameters.tTaskCycleTime := tPIDNutrientTaskCycleTime;
stPIDNutrientParameters.fKp := nPIDNutrientKp;
stPIDNutrientParameters.tTn := tPIDNutrientTn;
stPIDNutrientParameters.tTv := tPIDNutrientTv;
stPIDNutrientParameters.tTd := tPIDNutrientTd;
stPIDNutrientParameters.fOutMaxLimit := nPIDNutrientOutMaxLimit;
stPIDNutrientParameters.fOutMinLimit := nPIDNutrientOutMinLimit;
stPIDNutrientParameters.bPInTheFeedbackPath := bPIDNutrientPInTheFeedbackPath;
stPIDNutrientParameters.bDInTheFeedbackPath := bPIDNutrientDInTheFeedbackPath;
stPIDNutrientParameters.bARWOnIPartOnly := bPIDNutrientARWOnIPartOnly;

stPIDPHParameters.tCtrlCycleTime := tPIDPHCtrlCycleTime;
stPIDPHParameters.tTaskCycleTime := tPIDPHTaskCycleTime;
stPIDPHParameters.fKp := nPIDPHKp;
stPIDPHParameters.tTn := tPIDPHTn;
stPIDPHParameters.tTv := tPIDPHTv;
stPIDPHParameters.tTd := tPIDPHTd;
stPIDPHParameters.fOutMaxLimit := nPIDPHOutMaxLimit;
stPIDPHParameters.fOutMinLimit := nPIDPHOutMinLimit;
stPIDPHParameters.bPInTheFeedbackPath := bPIDPHPInTheFeedbackPath;
stPIDPHParameters.bDInTheFeedbackPath := bPIDPHDInTheFeedbackPath;
stPIDPHParameters.bARWOnIPartOnly := bPIDPHARWOnIPartOnly;
END_METHOD

END_FUNCTION_BLOCK

// ---- POUs/04 Control Loops/Dosing Machine/FB_ControlLoop_DissOx.TcPOU
(*
	Function Block which performs a level control using a DOL pump and a high level switch
*)
{attribute 'OPC.UA.DA.StructuredType' := '1'}
FUNCTION_BLOCK FB_ControlLoop_DissOx EXTENDS FB_BaseDevice
VAR_IN_OUT
	fbInjector: 			FB_OxygenInjector;
	fbSensorDissOx: 		FB_Sensor_AtlasDO;
	nSetPoint:				REAL;
END_VAR


VAR PERSISTENT
	tDebounce: TIME := T#1M; 
END_VAR

VAR
	bFirstRun: BOOL := TRUE;
	eSMState: (WAIT, DOSE_ON, DOSE_OFF, TURNING_OFF);
	fbTON_Debouce: TON := (PT := tDebounce, IN := FALSE);

END_VAR

IF bFirstRun THEN
	
	bFirstRun := FALSE;
END_IF


IF GVL.bAutoUpdateDeviceState THEN
	eState := eStateTarget;	
END_IF


IF eMode = E_DeviceMode.MANUAL OR eStateTarget = E_DeviceState.ON THEN
	bEnable := TRUE;
	fbInjector.enable();
END_IF

IF bEnable AND (eStateTarget = E_DeviceState.ON) AND (eSMState <> DOSE_ON) THEN
		eSMState := DOSE_OFF;
		fbInjector.enable();
END_IF


IF (bEnable = FALSE) OR (eStateTarget = E_DeviceState.OFF) THEN
		eSMState := TURNING_OFF;
		fbInjector.disable();
END_IF


IF bEnable THEN
	CASE eSMState OF
		WAIT:
			// Do nothing
			eState := E_DeviceState.OFF;
			
			
		DOSE_OFF:
			fbTON_Debouce(PT := tDebounce, IN := TRUE);
			eState := E_DeviceState.ON;
			fbInjector.setCommand(StateTarget := E_DeviceState.OFF);
			IF (fbSensorDissOx.getValue() < nSetPoint)  AND (fbTON_Debouce.Q) THEN
				eSMState := DOSE_ON;
			END_IF
			
		DOSE_ON:
			fbTON_Debouce(IN := FALSE);
			eState := E_DeviceState.ON;
			fbInjector.setCommand(StateTarget := E_DeviceState.ON);
			IF (fbSensorDissOx.getValue() > nSetPoint)THEN
				eSMState := DOSE_OFF;
			END_IF
			
		TURNING_OFF:
			eState := E_DeviceState.TURNING_OFF;
			fbInjector.setCommand(StateTarget := E_DeviceState.OFF);
			eSMState := WAIT;
			
	END_CASE
END_IF

METHOD setState : BOOL
VAR_INPUT
	state : E_DeviceState;
END_VAR

eState := state;
END_METHOD

END_FUNCTION_BLOCK

// ---- POUs/04 Control Loops/Dosing Machine/FB_ControlLoop_Dosing.TcPOU
FUNCTION_BLOCK FB_ControlLoop_Dosing EXTENDS FB_BaseDevice

VAR PERSISTENT
	nVolumeWater: REAL := 200.0; // Litres
	
	nPHDownFactor: LREAL := 10000;
	nPH_ProcessValue_Moles: FLOAT;
	nPH_ProcessValue: FLOAT;
	nPH_Setpoint: FLOAT;
	nPH_LowBand: FLOAT;
	nPH_HighBand: FLOAT;
	
	nPHSensorValDummy: FLOAT;
	nNutrient_ProcessValue: FLOAT;
	
	{attribute 'OPC.UA.DA' := '0'} 
	eCurrentNutrient: 			(NUTRIENT_A,NUTRIENT_B,NUTRIENT_C, PH) := NUTRIENT_C;
	bPHOnly: BOOL := TRUE;
	
	nPIDNutrientMaxDoseRate: UINT;
	nPIDNutrientMinDoseRate: UINT;
	tPIDNutrientTimeBetweenDoses: TIME;
	nPIDPHMaxDoseRate: UINT;
	nPIDPHMinDoseRate: UINT;
	tPIDPHTimeBetweenDoses: TIME;
	
	benableDosPumps: BOOL := TRUE;
	{attribute 'OPC.UA.DA' := '1'} 
	tPIDLoopTime: TIME := T#1M;	//5 second PID calculation
	
	// PID loop variables below
	nPIDNutrientSetpoint:		REAL; 
	nPIDNutrientSetpointBand:	REAL; // %
	nPIDNutrientManSyncVal:		REAL;
	bPIDNutrientSync: 			BOOL;
	nPIDNutrientError:			REAL;
	nPIDNutrientErrorPerc:		REAL;  // this is used to check if we are at 75%
	nPIDNutrientOutput: 		LREAL; 
	bPIDNutrientHold: 			BOOL;
	ePIDNutrientMode: 			E_CTRL_MODE;
	stPIDNutrientParameters: 	ST_CTRL_PID_PARAMS;
	ePIDNutrientErrorId: 		E_CTRL_ERRORCODES;
	bPIDNutrientError: 			BOOL;
	bPIDNutrientARWactive: 		BOOL;
	
	//stPIDParams values
	tPIDNutrientCtrlCycleTime: 		TIME := tPIDLoopTime;
	tPIDNutrientTaskCycleTime:		TIME := T#10MS;
	nPIDNutrientKp:  				REAL := 1.0;
	nPIDNutrientCompensator:  		REAL := 1.0/1000.0;
	tPIDNutrientTn: 				TIME := T#0S;
	tPIDNutrientTv:					TIME := T#0S;
	tPIDNutrientTd:					TIME := T#200S; 
	nPIDNutrientOutMaxLimit: 		REAL := 300; 		// this is set in the cyclic routine, the error band moves with the setpoint
	nPIDNutrientOutMinLimit:		REAL := 0;
	bPIDNutrientPInTheFeedbackPath: BOOL := FALSE;
	bPIDNutrientDInTheFeedbackPath: BOOL := FALSE;
	bPIDNutrientARWOnIPartOnly:		BOOL := FALSE;
	
	
	
	// Inputs
	nPIDPHSetpoint_Moles:			FLOAT; 					// Setpoint of the controlled variable (units pH)
	nPIDPHSetpoint_HydrogenMoles:	FLOAT;			// Setpoint of the controlled variable (H+ moles)
	nPIDPHSetpointBand:		REAL;					// 
	nPIDPHManSyncVal:		REAL;					// 	Input, to whose value it is possible to set the internal state of the PID-element.
	bPIDPHSync: 			BOOL;					//  A rising edge at this input sets the PID-element to the value "fManSyncValue".
	nPIDPHError:			REAL;					//  This is abs(actual - setpoint)

	bPIDPHHold: 			BOOL;					// 	A TRUE at this input will hold the internal state (and therefore also the output) constant at its current value, independently of the control deviation.			
	ePIDPHMode: 			E_CTRL_MODE;			//  Input that specifies the operation mode of the function block.
	
	
	// Outputs 
	nPIDPHOutput: 			LREAL;					// Output of the PID element
	ePIDPHErrorId: 			E_CTRL_ERRORCODES;		// Supplies the error number when the output bError is set.
	bPIDPHError: 			BOOL;					// Becomes TRUE, as soon as an error occurs.
	bPIDPHARWactive: 		BOOL;					// A TRUE at this output indicates that the PID-element is being restricted.
	
	// Inputs & Outputs (VAR IN OUT)
	stPIDPHParameters: 		ST_CTRL_PID_PARAMS;		// Parameter structure of the PID element
	
	//stPIDParams values
	tPIDPHCtrlCycleTime: 		TIME := tPIDLoopTime;	// Cycle time with which the control loop is processed. This must be greater than or equal to the TaskCycleTime. The function block uses this input value to calculate internally whether the state and the output values have to be updated in the current cycle.
	tPIDPHTaskCycleTime:		TIME := T#10MS;	// Cycle TIME with which the FUNCTION block is called. IF the FUNCTION block is called in every cycle THIS corresponds TO the task cycle TIME OF the calling task
	nPIDPHKp:  					FLOAT := 16327.71;	// Controller amplification / controller coefficient (our system gain is 0.0000025)
	tPIDPHTn: 					TIME := T#0S;  			// Integral action time; if this is parameterized to T#0s, the I component is deactivated.
	tPIDPHTv:					TIME := T#0S;  			// Derivative action time; if this is parameterized to T#0s, the D component is deactivated.
	tPIDPHTd:					TIME := T#200S; 		// Damping time
	nPIDPHOutMaxLimit: 			REAL := 300; 	// Upper limit at which integration is halted and to which the output is limited (ARW measure). Reaching this limit is indicated by a TRUE at the bARWActive output.
	nPIDPHOutMinLimit:			REAL := -300;		// 	Lower LIMIT AT which integration is halted AND TO which the output is limited (ARW measure). Reaching THIS LIMIT is indicated BY a TRUE AT the bARWActive output
	bPIDPHPInTheFeedbackPath: 	BOOL := FALSE;	// Input value of the internal P-element can be selected with this input (see functional diagram). Standard setting: FALSE
	bPIDPHDInTheFeedbackPath:	BOOL := FALSE;	//  Input value of the internal D-element can be selected with this input (see functional diagram). Standard setting: FALSE
	bPIDPHARWOnIPartOnly:		BOOL := FALSE;			// 	If this parameter is FALSE (the standard setting), the integration of the I-component is halted if the complete controller output reaches the upper or lower limit. If it is TRUE, the integration is halted if the I-component (the output of the integrator) reaches some limit. (Cf. functional diagram.)
	
	nPIDPH_Out: INT;
	tgNutrientOutLatch: R_TRIG;
	nNutrientOutput: LREAL := 0;
END_VAR

VAR
	bFirstRun: BOOL := TRUE;
	bResetTimer: BOOL := FALSE;
	
	{attribute 'OPC.UA.DA' := '0'} 
	fbSensor_EC:	I_Sensor(SensorID := '', SensorDescr := '' , SensorType := E_SensorType.Analogue);
	{attribute 'OPC.UA.DA' := '0'} 
	fbSensor_DO:	I_Sensor(SensorID := '', SensorDescr := '' , SensorType := E_SensorType.Analogue);
	{attribute 'OPC.UA.DA' := '0'} 
	fbSensor_ORP:	I_Sensor(SensorID := '', SensorDescr := '' , SensorType := E_SensorType.Analogue);
	{attribute 'OPC.UA.DA' := '0'} 
	fbSensor_PH:	I_Sensor(SensorID := '', SensorDescr := '' , SensorType := E_SensorType.Analogue);
	{attribute 'OPC.UA.DA' := '0'} 
	fbSensor_TEMP:	I_Sensor(SensorID := '', SensorDescr := '' , SensorType := E_SensorType.Analogue);	

	{attribute 'OPC.UA.DA' := '0'} 
	fbDosingPump_phUp:  		I_PumpDosing;
	{attribute 'OPC.UA.DA' := '0'} 
	fbDosingPump_phDOwn:  		I_PumpDosing;
	{attribute 'OPC.UA.DA' := '0'} 
	fbDosingPump_Nutrient_A:  	I_PumpDosing;
	{attribute 'OPC.UA.DA' := '0'} 
	fbDosingPump_Nutrient_B:  	I_PumpDosing;
	{attribute 'OPC.UA.DA' := '0'} 
	fbDosingPump_Nutrient_C:  	I_PumpDosing;
	{attribute 'OPC.UA.DA' := '0'} 
	eSMState: 					(WAIT, CALCULATE, NUTRIENT_ONLY, NUTRIENT_AND_PH, PH_ONLY) := WAIT;

	
	bDoseRequestSent:		BOOL := FALSE;
	bDoseRequestComplete: 	BOOL := FALSE;
	
	{attribute 'OPC.UA.DA' := '0'} 
	fbTON_PIDLoop: TON := (PT := tPIDLoopTime, IN := FALSE);
	
	{attribute 'OPC.UA.DA' := '0'}
	PID_Nutrient: FB_CTRL_PID;
	
	{attribute 'OPC.UA.DA' := '0'}
	PID_PH: FB_CTRL_PID;
	
	tgDisableOneShot: F_TRIG;
	
END_VAR

IF bFirstRun THEN
	fbTON_PIDLoop(PT := tPIDLoopTime, IN := TRUE);
	bFirstRun := FALSE;
END_IF


eState := eStateTarget;

IF fbTON_PIDLoop.Q THEN
	fbTON_PIDLoop.IN := FALSE;
	eSMState := CALCULATE;		// This is the entry point to start PID calculations and dosing
END_IF

fbTON_PIDLoop(PT := tPIDLoopTime);

calcInput();
updatePIDParams();
calcError();
tgNutrientOutLatch();
tgDisableOneShot(CLK := bEnable);

IF nPIDNutrientSetpoint > -1 THEN
	IF nPIDNutrientError > 0 THEN
		nPIDNutrientErrorPerc:=	1 - (ABS(nPIDNutrientError)/(nPIDNutrientSetpoint)); // this is used to decide if we opt for nutrient only dosing or nutrient and PH
	ELSE
		nPIDNutrientErrorPerc := 1; //
	END_IF
END_IF

IF eState = E_DeviceState.ON AND bEnable THEN
	//IF (nPH_ProcessValue < nPH_LowBand) OR (nPH_ProcessValue > nPH_HighBand) THEN
	PID_PH(		fSetpointValue := nPIDPHSetpoint_Moles, 			fActualValue := nPH_ProcessValue_Moles, 			stParams := stPIDPHParameters); //, eMode := E_CTRL_MODE.eCTRL_MODE_ACTIVE);	
	//END_IF
	
	PID_Nutrient(	fSetpointValue := nPIDNutrientSetpoint, 	fActualValue := nNutrient_ProcessValue, 	stParams := stPIDNutrientParameters);//, eMode := E_CTRL_MODE.eCTRL_MODE_ACTIVE);
END_IF

IF bEnable AND benableDosPumps AND (eState = E_DeviceState.ON) THEN
	fbDosingPump_Nutrient_A.enable();
	fbDosingPump_Nutrient_B.enable();
	fbDosingPump_Nutrient_C.enable();
	fbDosingPump_phDOwn.enable();
	fbDosingPump_phUp.enable();
	//fbDosingPump_phUp.disable();   // temporarily disable pH up dosing 
END_IF

IF tgDisableOneShot.Q THEN   // handle the case where the control lloop is turned off mid-dose
	fbDosingPump_Nutrient_A.setOFF(RequestComplete := 0);
	fbDosingPump_Nutrient_B.setOFF(RequestComplete := 0);
	fbDosingPump_Nutrient_C.setOFF(RequestComplete := 0);
	fbDosingPump_phDOwn.setOFF(RequestComplete := 0);
	fbDosingPump_phUp.setOFF(RequestComplete := 0);
	fbDosingPump_Nutrient_A.disable();
	fbDosingPump_Nutrient_B.disable();
	fbDosingPump_Nutrient_C.disable();
	fbDosingPump_phDOwn.disable();
	fbDosingPump_phUp.disable();
	eStateTarget := E_DeviceState.OFF;
	PID_Nutrient.eMode := E_CTRL_MODE.eCTRL_MODE_RESET;
	PID_PH.eMode := E_CTRL_MODE.eCTRL_MODE_RESET;
END_IF


CASE eSMState OF

	WAIT:
		// Do nothing and wait for timer to trigger
		
	CALCULATE:
	
		IF (eStateTarget = E_DeviceState.ON) AND bEnable THEN 
			
			IF nPIDNutrientErrorPerc < 0.75 THEN    // only bring in pH when EC is 75% percent of setpoint
				eSMState := NUTRIENT_ONLY;
				//tPIDNutrientCtrlCycleTime := tPIDLoopTime * 3;
				tPIDNutrientCtrlCycleTime := tPIDNutrientTaskCycleTime;
				//PID_Nutrient.eMode 		:= E_CTRL_MODE.eCTRL_MODE_ACTIVE;
				PID_PH.eMode 			:= E_CTRL_MODE.eCTRL_MODE_RESET;

			ELSIF (nPIDNutrientError < 0.03) AND (eCurrentNutrient = PH) THEN
				
				eSMState := PH_ONLY;
				//tPIDPHCtrlCycleTime := tPIDLoopTime;
				tPIDPHCtrlCycleTime := tPIDPHTaskCycleTime;
				PID_Nutrient.eMode 		:= E_CTRL_MODE.eCTRL_MODE_RESET;
				//PID_PH.eMode 			:= E_CTRL_MODE.eCTRL_MODE_ACTIVE;
			ELSE 
				eSMState := NUTRIENT_AND_PH;
				//tPIDNutrientCtrlCycleTime := tPIDLoopTime * 4;
				tPIDNutrientCtrlCycleTime := tPIDNutrientTaskCycleTime;
				//tPIDPHCtrlCycleTime := tPIDLoopTime * 4;
				tPIDPHCtrlCycleTime := tPIDPHTaskCycleTime;
				//PID_Nutrient.eMode 		:= E_CTRL_MODE.eCTRL_MODE_ACTIVE;
				//PID_PH.eMode 			:= E_CTRL_MODE.eCTRL_MODE_ACTIVE;
			END_IF
		END_IF
		
		
		IF bPHOnly AND (eStateTarget = E_DeviceState.ON) THEN  // this was used for commissioning when we were only doing PH
			eSMState := PH_ONLY;
			fbDosingPump_phUp.enable();
			fbDosingPump_phDOwn.enable();
		END_IF
		
		IF eCurrentNutrient = NUTRIENT_A THEN
			tgNutrientOutLatch(CLK := TRUE);
		END_IF
		
		IF tgNutrientOutLatch.Q THEN
			nNutrientOutput := PID_Nutrient.fOut;
		END_IF
		
		fbTON_PIDLoop(IN := FALSE);
		
	NUTRIENT_AND_PH:
		// Activate both Nutrient and PH Loops
		PID_Nutrient.eMode 		:= E_CTRL_MODE.eCTRL_MODE_ACTIVE;
		
		nPIDPH_Out := LREAL_TO_INT(PID_PH.fOut); 
		
		IF (nPH_ProcessValue < nPH_LowBand) OR (nPH_ProcessValue > nPH_HighBand) THEN
				PID_PH.eMode 		:= E_CTRL_MODE.eCTRL_MODE_ACTIVE;
		ELSE
				PID_PH.eMode 		:= E_CTRL_MODE.eCTRL_MODE_RESET;	// reset the PID loop if we are inside the deadband to avoid integral wind-up
		END_IF
		
		
		// Execute the PID loop calculations
		//PID_PH(fSetpointValue := nPIDPHSetpoint_HydrogenMoles, fActualValue := nPH_ProcessValue, stParams := stPIDPHParameters);
		//PID_Nutrient(fSetpointValue := nPIDNutrientSetpoint, fActualValue := nNutrient_ProcessValue, stParams := stPIDNutrientParameters);
		
		CASE eCurrentNutrient OF
			NUTRIENT_A:
				fbDosingPump_Nutrient_A.executeDose(DoseQtyMls := LREAL_TO_UINT(nNutrientOutput), DoseRateMlph := 100, RequestComplete := 0, RequestAccepted => bDoseRequestComplete);
				eCurrentNutrient := NUTRIENT_B;
			NUTRIENT_B:
				fbDosingPump_Nutrient_B.executeDose(DoseQtyMls := LREAL_TO_UINT(nNutrientOutput), DoseRateMlph := 100, RequestComplete := 0, RequestAccepted => bDoseRequestComplete);
				eCurrentNutrient := NUTRIENT_C;
				tgNutrientOutLatch(CLK := FALSE);
			NUTRIENT_C:
				fbDosingPump_Nutrient_C.executeDose(DoseQtyMls := LREAL_TO_UINT(nNutrientOutput), DoseRateMlph := 100, RequestComplete := 0, RequestAccepted => bDoseRequestComplete);
				eCurrentNutrient := PH;
			PH:
				IF (nPH_ProcessValue < nPH_LowBand) OR (nPH_ProcessValue > nPH_HighBand) THEN
					IF nPIDPH_Out > 0 THEN
						fbDosingPump_phDOwn.executeDose(DoseQtyMls := (PID_PH.fOut/nPHDownFactor), DoseRateMlph := 100, RequestComplete := 0, RequestAccepted => bDoseRequestComplete);
					ELSIF nPIDPH_Out < 0 THEN
						fbDosingPump_phUp.executeDose(DoseQtyMls := ABS(PID_PH.fOut), DoseRateMlph := 100, RequestComplete := 0, RequestAccepted => bDoseRequestComplete);
					END_IF
				END_IF
				eCurrentNutrient := NUTRIENT_A;	
				
		END_CASE	
		eSMState := WAIT; // go back to wait for the next timer trigger
		fbTON_PIDLoop.IN := TRUE;			
		
			
		NUTRIENT_ONLY:
		
			PID_Nutrient.eMode := E_CTRL_MODE.eCTRL_MODE_ACTIVE;
			// Activate both Nutrient and PH Loops
			//PID_PH.eMode 			:= E_CTRL_MODE.eCTRL_MODE_IDLE; // E_CTRL_MODE.eCTRL_MODE_FREEZE; ----- <<<< FOR TESTING ONLY, PUT THIS BACK FOR DEPLOYMENT
			//PID_Nutrient.eMode 		:= E_CTRL_MODE.eCTRL_MODE_ACTIVE;
			
			// Execute the PID loop calculations
			//PID_Nutrient(fSetpointValue := nPIDNutrientSetpoint, fActualValue := nNutrient_ProcessValue, stParams := stPIDNutrientParameters, fOut => nNutrientOutput);
		
			CASE eCurrentNutrient OF
				PH:
					eCurrentNutrient := NUTRIENT_A;
				NUTRIENT_A:
					fbDosingPump_Nutrient_A.executeDose(DoseQtyMls := LREAL_TO_UINT(nNutrientOutput), DoseRateMlph := 100, RequestComplete := 0, RequestAccepted => bDoseRequestComplete);
					eCurrentNutrient := NUTRIENT_B;
				NUTRIENT_B:
					fbDosingPump_Nutrient_B.executeDose(DoseQtyMls := LREAL_TO_UINT(nNutrientOutput), DoseRateMlph := 100, RequestComplete := 0, RequestAccepted => bDoseRequestComplete);
					eCurrentNutrient := NUTRIENT_C;
					tgNutrientOutLatch(CLK := FALSE);
				NUTRIENT_C:
					fbDosingPump_Nutrient_C.executeDose(DoseQtyMls := LREAL_TO_UINT(nNutrientOutput), DoseRateMlph := 100, RequestComplete := 0, RequestAccepted => bDoseRequestComplete);
					eCurrentNutrient := NUTRIENT_A;
			END_CASE
			eSMState := WAIT; // go back to wait for the next timer trigger		
			fbTON_PIDLoop.IN := TRUE;	
			
			
		PH_ONLY:
		
			nPIDPH_Out := LREAL_TO_INT(PID_PH.fOut); 
			
			IF (nPH_ProcessValue < nPH_LowBand) OR (nPH_ProcessValue > nPH_HighBand) THEN
					PID_PH.eMode 		:= E_CTRL_MODE.eCTRL_MODE_ACTIVE;
			ELSE
					PID_PH.eMode 		:= E_CTRL_MODE.eCTRL_MODE_RESET;	// reset the PID loop if we are inside the deadband to avoid integral wind-up
			END_IF
			
			IF (nPH_ProcessValue < nPH_LowBand) OR (nPH_ProcessValue > nPH_HighBand) THEN
				IF nPIDPH_Out > 0 THEN
					fbDosingPump_phDOwn.executeDose(DoseQtyMls := (PID_PH.fOut/nPHDownFactor), DoseRateMlph := 100, RequestComplete := 0, RequestAccepted => bDoseRequestComplete);
				ELSIF nPIDPH_Out < 0 THEN
					fbDosingPump_phUp.executeDose(DoseQtyMls := ABS(PID_PH.fOut), DoseRateMlph := 100, RequestComplete := 0, RequestAccepted => bDoseRequestComplete);
				END_IF
			END_IF
			eCurrentNutrient := PH;	
		
			eSMState := WAIT; // go back to wait for the next timer trigger		
			fbTON_PIDLoop.IN := TRUE;			
			
END_CASE



IF NOT ((nPH_ProcessValue < nPH_LowBand) OR (nPH_ProcessValue > nPH_HighBand)) THEN
	PID_Nutrient.eMode := E_CTRL_MODE.eCTRL_MODE_RESET;
END_IF

METHOD calcError : BOOL
VAR_INPUT
END_VAR
nPIDNutrientError 	:= nPIDNutrientSetpoint - nNutrient_ProcessValue;
nPIDNutrientError 	:= nPIDNutrientError;

nPIDPHError			:= nPIDPHSetpoint_Moles - nPH_ProcessValue_Moles;
END_METHOD

METHOD calcInput : BOOL
VAR_INPUT
END_VAR
//nPIDPHSetpoint 			:= 	EXPT(10, -1.0 * fbSensor_PH.getValue());

nNutrient_ProcessValue 		:= 	fbSensor_EC.getValue();

//nPIDPHSetpoint 			:= 	EXPT(10, -1.0 * fbSensor_PH.getValue());

nPIDPHSetpoint_Moles		:= 	EXPT(10, -1.0 * nPH_Setpoint) * nVolumeWater;
nPH_ProcessValue_Moles		:= 	EXPT(10, -1.0 * fbSensor_PH.getValue())  * nVolumeWater;

nPH_ProcessValue			:= fbSensor_PH.getValue();
//nPH_Setpoint				:= fbSensor_PH.getValue();
// nPH_HighBand				:= nPH_Setpoint + 0.1;
nPH_HighBand				:= nPH_Setpoint;
nPH_LowBand					:= nPH_Setpoint - 0.07;
END_METHOD

METHOD FB_init : BOOL
VAR_INPUT
	bInitRetains : BOOL; // if TRUE, the retain variables are initialized (warm start / cold start)
	bInCopyCode : BOOL;  // if TRUE, the instance afterwards gets moved into the copy code (online change)
	
	DosingPump_phUp:  			I_PumpDosing;
	DosingPump_phDOwn:  		I_PumpDosing;
	DosingPump_Nutrient_A:  	I_PumpDosing;
	DosingPump_Nutrient_B:  	I_PumpDosing;
	DosingPump_Nutrient_C:  	I_PumpDosing;
	
	ID: STRING(80);
	Description: STRING(80);
	
	
	Sensor_EC:				I_Sensor(SensorID := '', SensorDescr := '' , SensorType := E_SensorType.Analogue);
	Sensor_DO:				I_Sensor(SensorID := '', SensorDescr := '' , SensorType := E_SensorType.Analogue);
	Sensor_ORP:				I_Sensor(SensorID := '', SensorDescr := '' , SensorType := E_SensorType.Analogue);
	Sensor_PH:				I_Sensor(SensorID := '', SensorDescr := '' , SensorType := E_SensorType.Analogue);
	Sensor_TEMP:			I_Sensor(SensorID := '', SensorDescr := '' , SensorType := E_SensorType.Analogue);
	
END_VAR
fbDosingPump_phUp := DosingPump_phUp;
fbDosingPump_phDOwn := DosingPump_phDOwn;
fbDosingPump_Nutrient_A := DosingPump_Nutrient_A;
fbDosingPump_Nutrient_B := DosingPump_Nutrient_B;
fbDosingPump_Nutrient_C := DosingPump_Nutrient_C;

fbSensor_EC := Sensor_EC;
fbSensor_DO := Sensor_DO;
fbSensor_ORP := Sensor_ORP;
fbSensor_PH := Sensor_PH;
fbSensor_TEMP := Sensor_TEMP;	
sID := ID;
sDescr := Description;
END_METHOD

METHOD setParams : BOOL
VAR_INPUT
	(*
	NutrientMaxDoseRate: UINT;
	NutrientMinDoseRate: UINT;
	NutrientTimeBetweenDoses: TIME;
	PHMaxDoseRate: UINT;
	PHMinDoseRate: UINT;
	PHTimeBetweenDoses: TIME;


	// PID loop variables below
	*)
	NutrientSetpoint:		REAL; 
	(*
	NutrientSetpointBand:	REAL;
	
	NutrientManSyncVal:		REAL;
	NutrientSync: 			BOOL; 
	NutrientHold: 			BOOL;
	NutrientMode: 			E_CTRL_MODE;
	NutrientCtrlCycleTime: 	TIME;
	NutrientTaskCycleTime:	TIME;
	
	//stPIDParams values
	NutrientKp:  				REAL;
	NutrientTn: 				TIME; 
	NutrientTv:					TIME; 
	NutrientTd:					TIME; 
	NutrientOutMaxLimit: 		REAL;
	NutrientOutMinLimit:		REAL;
	NutrientPInTheFeedbackPath: BOOL;
	NutrientDInTheFeedbackPath: BOOL;
	NutrientARWOnIPartOnly:		BOOL;
	
	*)
	PHSetpoint:			REAL; 
	PHSetpointBand:		REAL;
	(*
	PHManSyncVal:		REAL;
	PHSync: 			BOOL;
	PHHold: 			BOOL;
	PHMode: 			E_CTRL_MODE;
	PHCtrlCycleTime: 		TIME;
	PHTaskCycleTime:		TIME;
	
	
	//stPIDParams values
	*)
	PHKp:  					REAL;
	PHTn: 					TIME;
	PHTv:					TIME;
	PHTd:					TIME; 
	(*
	PHOutMaxLimit: 			REAL; 		
	PHOutMinLimit:			REAL;
	PHPInTheFeedbackPath: 	BOOL;
	PHDInTheFeedbackPath:	BOOL;
	PHARWOnIPartOnly:		BOOL;
	*)
	
END_VAR
(*
nPIDNutrientMaxDoseRate := 				NutrientMaxDoseRate;
nPIDNutrientMinDoseRate := 				NutrientMinDoseRate;
tPIDNutrientTimeBetweenDoses := 		NutrientTimeBetweenDoses;

nPIDPHMaxDoseRate := 					PHMaxDoseRate;
nPIDPHMinDoseRate := 					PHMinDoseRate;
tPIDPHTimeBetweenDoses := 				PHTimeBetweenDoses;

*)
nPIDNutrientSetpoint := 				NutrientSetpoint;
(*
nPIDNutrientSetpointBand := 			NutrientSetpointBand;
nPIDNutrientManSyncVal := 				NutrientManSyncVal;
bPIDNutrientSync := 					NutrientSync;
bPIDNutrientHold := 					NutrientHold;
ePIDNutrientMode := 					NutrientMode;
tPIDNutrientCtrlCycleTime := 			NutrientCtrlCycleTime;
tPIDNutrientTaskCycleTime := 			NutrientTaskCycleTime;

nPIDNutrientKp := 						NutrientKp;
tPIDNutrientTn := 						NutrientTn;
tPIDNutrientTv := 						NutrientTv;
tPIDNutrientTd := 						NutrientTd;
nPIDNutrientOutMaxLimit := 				NutrientOutMaxLimit;
nPIDNutrientOutMinLimit := 				NutrientOutMinLimit;
bPIDNutrientPInTheFeedbackPath := 		NutrientPInTheFeedbackPath;
bPIDNutrientDInTheFeedbackPath := 		NutrientDInTheFeedbackPath;
bPIDNutrientARWactive := 				NutrientARWOnIPartOnly;
*)
nPH_Setpoint := 						PHSetpoint;

nPIDPHSetpointBand := 					PHSetpointBand;
(*
nPIDPHManSyncVal := 					PHManSyncVal;
bPIDPHSync := 							PHSync;
bPIDPHHold := 							PHHold;
ePIDPHMode := 							PHMode;
tPIDPHCtrlCycleTime := 					PHCtrlCycleTime;
tPIDPHTaskCycleTime := 					PHTaskCycleTime;
*)
nPIDPHKp := 							PHKp;
tPIDPHTn := 							PHTn * 1000;
tPIDPHTv := 							PHTv * 1000;
tPIDPHTd := 							PHTd * 1000;
(*
nPIDPHOutMaxLimit := 					PHOutMaxLimit;
nPIDPHOutMinLimit := 					PHOutMinLimit;
bPIDPHPInTheFeedbackPath := 			PHPInTheFeedbackPath;
bPIDPHDInTheFeedbackPath := 			PHDInTheFeedbackPath;
bPIDPHARWactive := 						PHARWOnIPartOnly;
*)
END_METHOD

METHOD updatePIDParams : BOOL
VAR_INPUT
END_VAR
stPIDNutrientParameters.tCtrlCycleTime := tPIDNutrientCtrlCycleTime;
stPIDNutrientParameters.tTaskCycleTime := tPIDNutrientTaskCycleTime;
stPIDNutrientParameters.fKp := nPIDNutrientKp;
stPIDNutrientParameters.tTn := tPIDNutrientTn;
stPIDNutrientParameters.tTv := tPIDNutrientTv;
stPIDNutrientParameters.tTd := tPIDNutrientTd;
stPIDNutrientParameters.fOutMaxLimit := nPIDNutrientOutMaxLimit;
stPIDNutrientParameters.fOutMinLimit := nPIDNutrientOutMinLimit;
stPIDNutrientParameters.bPInTheFeedbackPath := bPIDNutrientPInTheFeedbackPath;
stPIDNutrientParameters.bDInTheFeedbackPath := bPIDNutrientDInTheFeedbackPath;
stPIDNutrientParameters.bARWOnIPartOnly := bPIDNutrientARWOnIPartOnly;

stPIDPHParameters.tCtrlCycleTime := tPIDPHCtrlCycleTime;
stPIDPHParameters.tTaskCycleTime := tPIDPHTaskCycleTime;
stPIDPHParameters.fKp := nPIDPHKp;
stPIDPHParameters.tTn := tPIDPHTn;
stPIDPHParameters.tTv := tPIDPHTv;
stPIDPHParameters.tTd := tPIDPHTd;
stPIDPHParameters.fOutMaxLimit := nPIDPHOutMaxLimit;
stPIDPHParameters.fOutMinLimit := nPIDPHOutMinLimit;
stPIDPHParameters.bPInTheFeedbackPath := bPIDPHPInTheFeedbackPath;
stPIDPHParameters.bDInTheFeedbackPath := bPIDPHDInTheFeedbackPath;
stPIDPHParameters.bARWOnIPartOnly := bPIDPHARWOnIPartOnly;
END_METHOD

END_FUNCTION_BLOCK

// ---- POUs/04 Control Loops/Dosing Machine/FB_ControlLoop_HVAC.TcPOU
(*
	Function Block which performs a bang-bang control loop.
*)
{attribute 'OPC.UA.DA.StructuredType' := '1'}
FUNCTION_BLOCK FB_ControlLoop_HVAC EXTENDS FB_BaseDevice
VAR_INPUT PERSISTENT

	{attribute 'OPC.UA.DA' := '1'}
	nProcessValue : REAL;  
	{attribute 'OPC.UA.DA' := '1'}
	rSetpoint: REAL;

	{attribute 'OPC.UA.DA' := '1'}
	rAlarmHigh : REAL;
	{attribute 'OPC.UA.DA' := '1'}
	rAlarmLow : REAL;
	{attribute 'OPC.UA.DA' := '1'}
	rLimitHigh : REAL; // the upper limit of the desirable range (when the downward adjustment is activated)
	{attribute 'OPC.UA.DA' := '1'}
	rLimitLow : REAL; // lower limit of the desirable range (when the upward adjustment is activated)
	{attribute 'OPC.UA.DA' := '1'}
	nAdjustDelay : INT := 30; // min time in seconds between adjustments
	{attribute 'OPC.UA.DA' := '1'}
	nAdjustDownIncrement : REAL := 0.5;
	{attribute 'OPC.UA.DA' := '1'}
	nAdjustUpIncrement : REAL := 0.5; 
	{attribute 'OPC.UA.DA' := '1'}
	rCurrentValue : REAL; 
	{attribute 'OPC.UA.DA' := '1'}
	bEnabled : BOOL; 
	{attribute 'OPC.UA.DA' := '1'}
	sParameterName : STRING;
	
	{attribute 'OPC.UA.DA' := '1'}
	nControlValue: POINTER TO REAL;
	{attribute 'OPC.UA.DA' := '1'}
	nControlValueCopy: REAL;
	
	{attribute 'OPC.UA.DA' := '1'} 
	tPIDLoopTime: TIME := T#1M;	// how often the PID loop should be executed
	
	
	{attribute 'OPC.UA.DA' := '1'}
	Mode:    E_CTRL_MODE;
END_VAR

VAR_OUTPUT

	{attribute 'OPC.UA.DA' := '1'}
	bAlarmHigh : BOOL;
	{attribute 'OPC.UA.DA' := '1'}
	bAlarmLow : BOOL;
END_VAR

VAR
	bFirstRun : BOOL;
	bResetTimer: BOOL := FALSE;
	tAdjustDownTimer : TON;
	tAdjustUpTimer : TON;
	tAdjustDelayTimer : TON;
	bAdjustDownActive : BOOL;
	bAdjustUpActive : BOOL;
	bDelayActive : BOOL;
	
	{attribute 'OPC.UA.DA' := '0'} 
	fbTON_PIDLoop: TON := (PT := tPIDLoopTime, IN := FALSE);
	
	{attribute 'OPC.UA.DA' := '0'}
	PID: FB_CTRL_PID;
	
	eSMState: 	(WAIT, CALCULATE, TRIG_UP, TRIG_DOWN) := WAIT;

END_VAR



VAR PERSISTENT

	n_ProcessValue: FLOAT;
	
	// PID loop variables below
	nPID_Setpoint:			REAL; 
	nPID_SetpointBand:		REAL; 
	nPID_ManSyncVal:		REAL;
	bPID_Sync: 				BOOL;
	nPID_Error:				REAL;
	nPID_ErrorPerc:			REAL;  
	nPID_Output: 			LREAL; 
	bPID_Hold: 				BOOL;
	ePID_Mode: 				E_CTRL_MODE;
	stPID_Parameters: 		ST_CTRL_PID_PARAMS;
	ePID_ErrorId: 			E_CTRL_ERRORCODES;
	bPID_Error: 			BOOL;
	bPID_ARWactive: 		BOOL;
	
	//stPIDParams values
	tPID_CtrlCycleTime: 		TIME := tPIDLoopTime;
	tPID_TaskCycleTime:			TIME := T#10MS;
	nPID_Kp:  					REAL := 1.0;
	nPID_Compensator:  			REAL := 1.0/1000.0;
	tPID_Tn: 					TIME := T#0S;
	tPID_Tv:					TIME := T#0S;
	tPID_Td:					TIME := T#200S; 
	nPID_OutMaxLimit: 			REAL := 300; 		// this is set in the cyclic routine, the error band moves with the setpoint
	nPID_OutMinLimit:			REAL := 0;
	bPID_PInTheFeedbackPath: 	BOOL := FALSE;
	bPID_DInTheFeedbackPath: 	BOOL := FALSE;
	bPID_ARWOnIPartOnly:		BOOL := FALSE;
	
	n_Output: LREAL := 0;
	
END_VAR

IF bFirstRun THEN
	fbTON_PIDLoop(PT := tPIDLoopTime, IN := TRUE);
	bFirstRun := FALSE;
END_IF

//eState := eStateTarget;

IF (NOT bEnable) OR (eState = E_DeviceState.IDLE) THEN
	eState := E_DeviceState.IDLE;
	eStateTarget := E_DeviceState.IDLE;
	PID.eMode := E_CTRL_MODE.eCTRL_MODE_RESET;
END_IF

IF bEnable AND (eState = E_DeviceState.RUNNING) THEN
	PID.eMode := E_CTRL_MODE.eCTRL_MODE_ACTIVE;
END_IF 


fbTON_PIDLoop(PT := tPIDLoopTime);
updatePIDParams();

nPID_Setpoint := (rLimitHigh + rLimitLow) / 2.0;
rSetpoint := (rLimitHigh + rLimitLow) / 2.0;
nPID_Error 	:= nPID_Setpoint - rCurrentValue; 


IF eState = E_DeviceState.RUNNING THEN
	PID( fSetpointValue := nPID_Setpoint, fActualValue := rCurrentValue, stParams := stPID_Parameters);
END_IF


// IF control loop is ON and the loop timer has elapsed then enter the calculate / action state machine below
IF fbTON_PIDLoop.Q  AND (eState = E_DeviceState.RUNNING) THEN
	fbTON_PIDLoop.IN 	:= FALSE;
	eSMState 			:= CALCULATE;		
END_IF


CASE eSMState OF

	WAIT:
		fbTON_PIDLoop(IN := TRUE);
	
	CALCULATE:
	
		IF (nPID_Setpoint >= 16) AND (nPID_Setpoint <= 32) THEN
			nControlValue^ := nPID_Setpoint;
		ELSIF (nPID_Setpoint < 16) THEN
			nControlValue^ := 16;
			
		ELSIF (nPID_Setpoint > 32) THEN
			nControlValue^ := 32;
		END_IF
		nControlValueCopy := nControlValue^;
	(*
		IF ABS((nControlValue^ - nPID_Setpoint) > 0.2) THEN
			nControlValue^ := nControlValue^ + PID.fOut;
		ELSE
			tPID_Tn := T#0S;
		END_IF
		// nControlValue^ :=  PID.fOut;
		
		IF nControlValue^ < 16 THEN
			nControlValue^ := 16;
		ELSIF nControlValue^ > 32 THEN
			nControlValue^ := 32;
		END_IF
		
		fbTON_PIDLoop(IN := FALSE);
		eSMState := WAIT;	
		
		*)
END_CASE

METHOD setState : BOOL
VAR_INPUT
	state : E_DeviceState;
END_VAR

eState := state;
END_METHOD


(*
	Run the timers for delay, adjust up and adjust down
*)
METHOD timers : BOOL
VAR_INPUT
END_VAR
tAdjustDelayTimer(IN := bDelayActive, PT := INT_TO_TIME(nAdjustDelay) * 1000);


IF tAdjustDelayTimer.Q THEN
	// the delay timer is finished so check if we need to activate an adjustment
	
	//bAdjustDownActive := (rCurrentValue > rLimitHigh);
	//bAdjustUpActive := (rCurrentValue < rLimitLow);
	
	bAdjustDownActive := (rCurrentValue > ((rLimitHigh + rLimitLow)/2.0)+0.6);
	bAdjustUpActive := (rCurrentValue < ((rLimitHigh + rLimitLow)/2.0)-0.6);
	
END_IF

// run the delay timer whenever we are not activating an output
bDelayActive := NOT bAdjustDownActive AND NOT bAdjustUpActive;
END_METHOD

METHOD updatePIDParams : BOOL
VAR_INPUT
END_VAR


stPID_Parameters.tCtrlCycleTime := 		tPID_CtrlCycleTime;
stPID_Parameters.tTaskCycleTime := 		tPID_TaskCycleTime;
stPID_Parameters.fKp := 				nPID_Kp;
stPID_Parameters.tTn := 				tPID_Tn;
stPID_Parameters.tTv := 				tPID_Tv;
stPID_Parameters.tTd := 				tPID_Td;
stPID_Parameters.fOutMaxLimit := 		nPID_OutMaxLimit;
stPID_Parameters.fOutMinLimit := 		nPID_OutMinLimit;
stPID_Parameters.bPInTheFeedbackPath := bPID_PInTheFeedbackPath;
stPID_Parameters.bDInTheFeedbackPath := bPID_DInTheFeedbackPath;
stPID_Parameters.bARWOnIPartOnly := 	bPID_ARWOnIPartOnly;
END_METHOD

END_FUNCTION_BLOCK

// ---- POUs/04 Control Loops/Dosing Machine/FB_ControlLoop_HVAC_1.TcPOU
(*
	Function Block which performs a bang-bang control loop.
*)
{attribute 'OPC.UA.DA.StructuredType' := '1'}
FUNCTION_BLOCK FB_ControlLoop_HVAC_1 EXTENDS FB_BaseDevice
VAR_INPUT PERSISTENT

	{attribute 'OPC.UA.DA' := '1'}
	nProcessValue : REAL;  
	{attribute 'OPC.UA.DA' := '1'}
	rSetpoint: REAL;

	{attribute 'OPC.UA.DA' := '1'}
	rAlarmHigh : REAL;
	{attribute 'OPC.UA.DA' := '1'}
	rAlarmLow : REAL;
	{attribute 'OPC.UA.DA' := '1'}
	rLimitHigh : REAL; // the upper limit of the desirable range (when the downward adjustment is activated)
	{attribute 'OPC.UA.DA' := '1'}
	rLimitLow : REAL; // lower limit of the desirable range (when the upward adjustment is activated)
	{attribute 'OPC.UA.DA' := '1'}
	nAdjustDelay : INT := 30; // min time in seconds between adjustments
	{attribute 'OPC.UA.DA' := '1'}
	nAdjustDownIncrement : REAL := 0.5;
	{attribute 'OPC.UA.DA' := '1'}
	nAdjustUpIncrement : REAL := 0.5; 
	{attribute 'OPC.UA.DA' := '1'}
	rCurrentValue : REAL; 
	{attribute 'OPC.UA.DA' := '1'}
	bEnabled : BOOL; 
	{attribute 'OPC.UA.DA' := '1'}
	sParameterName : STRING;
	
	{attribute 'OPC.UA.DA' := '1'}
	nControlValue: POINTER TO REAL;
	{attribute 'OPC.UA.DA' := '1'}
	nControlValueCopy: REAL;
	
	{attribute 'OPC.UA.DA' := '1'} 
	tPIDLoopTime: TIME := T#1M;	// how often the PID loop should be executed
	
	nStepChange: REAL;
	nDegPerHr: REAL;

	
	
	{attribute 'OPC.UA.DA' := '1'}
	Mode:    E_CTRL_MODE;
END_VAR

VAR_OUTPUT

	{attribute 'OPC.UA.DA' := '1'}
	bAlarmHigh : BOOL;
	{attribute 'OPC.UA.DA' := '1'}
	bAlarmLow : BOOL;
END_VAR

VAR
	bFirstRun : BOOL;
	bResetTimer: BOOL := FALSE;
	tAdjustDownTimer : TON;
	tAdjustUpTimer : TON;
	tAdjustDelayTimer : TON;
	bAdjustDownActive : BOOL;
	bAdjustUpActive : BOOL;
	bDelayActive : BOOL;
	
	{attribute 'OPC.UA.DA' := '0'} 
	fbTON_PIDLoop: TON := (PT := tPIDLoopTime, IN := FALSE);
	
	{attribute 'OPC.UA.DA' := '0'}
	PID: FB_CTRL_PID;
	
	eSMState: 	(WAIT, CALCULATE, TRIG_UP, TRIG_DOWN) := WAIT;

END_VAR



VAR PERSISTENT

	n_ProcessValue: FLOAT;
	
	// PID loop variables below
	nPID_Setpoint:			REAL; 
	nPID_SetpointBand:		REAL; 
	nPID_ManSyncVal:		REAL;
	bPID_Sync: 				BOOL;
	nPID_Error:				REAL;
	nPID_ErrorPerc:			REAL;  
	nPID_Output: 			LREAL; 
	bPID_Hold: 				BOOL;
	ePID_Mode: 				E_CTRL_MODE;
	stPID_Parameters: 		ST_CTRL_PID_PARAMS;
	ePID_ErrorId: 			E_CTRL_ERRORCODES;
	bPID_Error: 			BOOL;
	bPID_ARWactive: 		BOOL;
	
	//stPIDParams values
	tPID_CtrlCycleTime: 		TIME := tPIDLoopTime;
	tPID_TaskCycleTime:			TIME := T#10MS;
	nPID_Kp:  					REAL := 1.0;
	nPID_Compensator:  			REAL := 1.0/1000.0;
	tPID_Tn: 					TIME := T#0S;
	tPID_Tv:					TIME := T#0S;
	tPID_Td:					TIME := T#200S; 
	nPID_OutMaxLimit: 			REAL := 300; 		// this is set in the cyclic routine, the error band moves with the setpoint
	nPID_OutMinLimit:			REAL := 0;
	bPID_PInTheFeedbackPath: 	BOOL := FALSE;
	bPID_DInTheFeedbackPath: 	BOOL := FALSE;
	bPID_ARWOnIPartOnly:		BOOL := FALSE;
	
	n_Output: LREAL := 0;
	
	nDeadBandPerc: REAL := 0.05; 
	
END_VAR

IF bFirstRun THEN
	fbTON_PIDLoop(PT := tPIDLoopTime, IN := TRUE);
	bFirstRun := FALSE;
END_IF

//eState := eStateTarget;

IF (NOT bEnable) OR (eState = E_DeviceState.IDLE) THEN
	eState := E_DeviceState.IDLE;
	eStateTarget := E_DeviceState.IDLE;
	PID.eMode := E_CTRL_MODE.eCTRL_MODE_RESET;
END_IF

IF bEnable AND (eState = E_DeviceState.RUNNING) THEN
	PID.eMode := E_CTRL_MODE.eCTRL_MODE_ACTIVE;
END_IF 


fbTON_PIDLoop(PT := tPIDLoopTime);
updatePIDParams();

nPID_Setpoint := (rLimitHigh + rLimitLow) / 2.0;
rSetpoint := (rLimitHigh + rLimitLow) / 2.0;
nPID_Error 	:= nPID_Setpoint - rCurrentValue; 


IF eState = E_DeviceState.RUNNING THEN
	PID( fSetpointValue := nPID_Setpoint, fActualValue := rCurrentValue, stParams := stPID_Parameters);
END_IF


// IF control loop is ON and the loop timer has elapsed then enter the calculate / action state machine below
IF fbTON_PIDLoop.Q  AND (eState = E_DeviceState.RUNNING) THEN
	fbTON_PIDLoop.IN 	:= FALSE;
	eSMState 			:= CALCULATE;		
END_IF


CASE eSMState OF

	WAIT:
		fbTON_PIDLoop(IN := TRUE);
	
	CALCULATE:
		
		
		
		IF (rCurrentValue > (nPID_Setpoint * ( 1 + nDeadBandPerc))) THEN
			nControlValue^ := nControlValue^ - (nDegPerHr * (TIME_TO_LREAL(tPIDLoopTime)/3600000));
		ELSIF (rCurrentValue < (nPID_Setpoint * ( 1 - nDeadBandPerc))) THEN
			nControlValue^ := nControlValue^ + (nDegPerHr * (TIME_TO_LREAL(tPIDLoopTime)/3600000));
		END_IF
		
		IF nControlValue^ < 16 THEN
			nControlValue^ := 16;
		ELSIF nControlValue^ > 32 THEN
			nControlValue^ := 32;
		END_IF
		
		nControlValueCopy := nControlValue^;
		
		eSMState := WAIT;
		fbTON_PIDLoop(IN := FALSE);
 
	(*
		IF ABS((nControlValue^ - nPID_Setpoint) > 0.2) THEN
			nControlValue^ := nControlValue^ + PID.fOut;
		ELSE
			tPID_Tn := T#0S;
		END_IF
		// nControlValue^ :=  PID.fOut;
		
		IF nControlValue^ < 16 THEN
			nControlValue^ := 16;
		ELSIF nControlValue^ > 32 THEN
			nControlValue^ := 32;
		END_IF
		
		fbTON_PIDLoop(IN := FALSE);
		eSMState := WAIT;	
		
		*)
END_CASE

METHOD setState : BOOL
VAR_INPUT
	state : E_DeviceState;
END_VAR

eState := state;
END_METHOD


(*
	Run the timers for delay, adjust up and adjust down
*)
METHOD timers : BOOL
VAR_INPUT
END_VAR
tAdjustDelayTimer(IN := bDelayActive, PT := INT_TO_TIME(nAdjustDelay) * 1000);


IF tAdjustDelayTimer.Q THEN
	// the delay timer is finished so check if we need to activate an adjustment
	
	//bAdjustDownActive := (rCurrentValue > rLimitHigh);
	//bAdjustUpActive := (rCurrentValue < rLimitLow);
	
	bAdjustDownActive := (rCurrentValue > ((rLimitHigh + rLimitLow)/2.0)+0.6);
	bAdjustUpActive := (rCurrentValue < ((rLimitHigh + rLimitLow)/2.0)-0.6);
	
END_IF

// run the delay timer whenever we are not activating an output
bDelayActive := NOT bAdjustDownActive AND NOT bAdjustUpActive;
END_METHOD

METHOD updatePIDParams : BOOL
VAR_INPUT
END_VAR


stPID_Parameters.tCtrlCycleTime := 		tPID_CtrlCycleTime;
stPID_Parameters.tTaskCycleTime := 		tPID_TaskCycleTime;
stPID_Parameters.fKp := 				nPID_Kp;
stPID_Parameters.tTn := 				tPID_Tn;
stPID_Parameters.tTv := 				tPID_Tv;
stPID_Parameters.tTd := 				tPID_Td;
stPID_Parameters.fOutMaxLimit := 		nPID_OutMaxLimit;
stPID_Parameters.fOutMinLimit := 		nPID_OutMinLimit;
stPID_Parameters.bPInTheFeedbackPath := bPID_PInTheFeedbackPath;
stPID_Parameters.bDInTheFeedbackPath := bPID_DInTheFeedbackPath;
stPID_Parameters.bARWOnIPartOnly := 	bPID_ARWOnIPartOnly;
END_METHOD

END_FUNCTION_BLOCK

// ---- POUs/04 Control Loops/Dosing Machine/FB_ControlLoop_MainPumpPressure.TcPOU
FUNCTION_BLOCK FB_ControlLoop_MainPumpPressure

VAR
	{attribute 'OPC.UA.DA' := '0'}
	fbMainPump:  		I_PumpVSD;
	
	eSMState: 					(INIT, WAIT_TRIG, WAIT, CALCULATE) := INIT;
	
	eState_MaxHeadofOpenValve:  	(RECIRC, L1, L2, L3, L4, L5, L6, L7, L8, L9 , L10, L11, L12, L13, L14, L15, L16, L17, L18, L19, L20) := L1;
	bEnabled: BOOL := TRUE;
	bError: BOOL := FALSE;
	
	{attribute 'OPC.UA.DA' := '0'}
	fbTON_LoopTime: TON := (PT := T#1S);
	
END_VAR

VAR_IN_OUT
	setPointPressure: UINT := 0; // kPa 
	
END_VAR

fbTON_LoopTime();

CASE eSmstate OF
	
	INIT:

		eSMState := WAIT_TRIG;

	WAIT_TRIG:
	
		eSMState := WAIT;
	
	WAIT:
		IF fbTON_LoopTime.Q THEN
			fbTON_LoopTime(IN := FALSE);
			eSMState := CALCULATE;
		END_IF

	CALCULATE:
	
		IF eState_MaxHeadofOpenValve = RECIRC THEN
			setPointPressure := 200;
		ELSE
			CASE eState_MaxHeadofOpenValve OF
				L1: 
					setPointPressure := 270;
				L2: 
					setPointPressure := 340;
				L3: 
					setPointPressure := 410;
				L4: 
					setPointPressure := 480;
				L5: 
					setPointPressure := 550;
				L6: 
					setPointPressure := 620;
				L7: 
					setPointPressure := 690;
				L8: 
					setPointPressure := 760;
				L9: 
					setPointPressure := 830;
				L10: 
					setPointPressure := 900;
				L11: 
					setPointPressure := 970;
				L12: 
					setPointPressure := 1040;
				L13: 
					setPointPressure := 1100;
				L14: 
					setPointPressure := 1180;
				L15: 
					setPointPressure := 1250;
				L16: 
					setPointPressure := 1320;
				L17: 
					setPointPressure := 1390;
				L18: 
					setPointPressure := 1460;
				L19: 
					setPointPressure := 1530;
				L20: 
					setPointPressure := 1600;
				
			END_CASE
		END_IF
						

		eSMState := WAIT_TRIG;
END_CASE

METHOD FB_init : BOOL
VAR_INPUT
	bInitRetains : BOOL; // if TRUE, the retain variables are initialized (warm start / cold start)
	bInCopyCode : BOOL;  // if TRUE, the instance afterwards gets moved into the copy code (online change)
	
	MainPump:  		I_PumpVSD;
	
END_VAR
fbMainPump := MainPump;
END_METHOD

METHOD setCurrentLevel : BOOL
VAR_INPUT
	HighestLevel: UINT;
END_VAR

eState_MaxHeadofOpenValve := HighestLevel;
END_METHOD

END_FUNCTION_BLOCK

// ---- POUs/04 Control Loops/Dosing Machine/FB_ControlLoop_pH.TcPOU
FUNCTION_BLOCK FB_ControlLoop_pH

VAR
	fbDosingPump_phUp:  		I_PumpDosing;
	fbDosingPump_phDOwn:  		I_PumpDosing;	
	{attribute 'OPC.UA.DA' := '0'} 
	fbSensor_PH:	I_Sensor(SensorID := '', SensorDescr := '' , SensorType := E_SensorType.Analogue);
	{attribute 'OPC.UA.DA' := '0'} 
	fbSensor_TEMP:	I_Sensor(SensorID := '', SensorDescr := '' , SensorType := E_SensorType.Analogue);	
	
	eSMState: 					(INIT, WAIT_TRIG, WAIT, CALCULATE) := INIT;
	eCurrentNutrient: 			(PH) := PH;

	bEnabled: BOOL := TRUE;
	bError: BOOL := FALSE;
	
	bDoseRequestSent:		BOOL := FALSE;
	bDoseRequestComplete: 	BOOL := FALSE;
	
	{attribute 'OPC.UA.DA' := '0'}
	fbTON_PIDLoop: TON;
	tPIDLoopTime: TIME := T#5S;			//5 second PID calculation
	
	nPIDPHMaxDoseRate: UINT;
	nPIDPHMinDoseRate: UINT;
	tPIDPHTimeBetweenDoses: TIME;
	
		
	nPIDPHSetpoint:			REAL; 
	nPIDPHSetpointBand:		REAL := 0.05; // %
	nPIDPHManSyncVal:		REAL;
	bPIDPHSync: 			BOOL;
	nPIDPHError:			REAL;
	nPIDPHOutput: 			LREAL;
	bPIDPHHold: 			BOOL;
	ePIDPHMode: 			E_CTRL_MODE;
	stPIDPHParameters: 		ST_CTRL_PID_PARAMS;
	ePIDPHErrorId: 			E_CTRL_ERRORCODES;
	bPIDPHError: 			BOOL;
	bPIDPHARWactive: 		BOOL;
		
	//stPIDParams values
	tPIDPHCtrlCycleTime: 		TIME := T#5000MS;
	tPIDPHTaskCycleTime:		TIME := T#10MS;
	nPIDPHKp:  					REAL := 500.0;
	tPIDPHTn: 					TIME := T#0MS; 
	tPIDPHTv:					TIME := T#0MS; 
	tPIDPHTd:					TIME := T#0MS; 
	nPIDPHOutMaxLimit: 			REAL := 1E38; 		
	nPIDPHOutMinLimit:			REAL := -1E38;
	bPIDPHPInTheFeedbackPath: 	BOOL := FALSE;
	bPIDPHDInTheFeedbackPath:	BOOL := FALSE;
	bPIDPHARWOnIPartOnly:		BOOL := FALSE;
	
	{attribute 'OPC.UA.DA' := '0'}
	PID_PH: FB_CTRL_PID;
	
END_VAR



CASE eSMState OF
	
	INIT:
		initPIDLoops();
		eSMState := WAIT_TRIG;

	WAIT_TRIG:
	
		fbTON_PIDLoop(IN:= TRUE, PT := tPIDLoopTime); // this controls the PID control loop cycle time
		nPIDPHError:= nPIDPHSetpoint - fbSensor_PH.getValue();
		eSMState := WAIT;
	
	WAIT:
		IF fbTON_PIDLoop.Q THEN
			fbTON_PIDLoop(IN := FALSE);
			eSMState := CALCULATE;
		END_IF

	CALCULATE:
						
		PID_PH(			fSetpointValue		:= nPIDPHSetpoint,
						fActualValue		:= fbSensor_PH.getValue(),
						fManSyncValue		:= nPIDPHManSyncVal,
						bSync				:= bPIDPHSync,
						eMode				:= ePIDPHMode,
						bHold				:= bPIDPHHold,
						stParams			:= stPIDPHParameters,
						fOut				=> nPIDPHOutput,
						bARWactive			=> bPIDPHARWactive,
						eErrorId			=> ePIDPHErrorId,
						bError				=> bPIDPHError );

		IF nPIDPHError > 0 AND bDoseRequestSent = FALSE THEN
			fbDosingPump_phUp.executeDose(DoseQtyMls := LREAL_TO_UINT(nPIDPHOutput), DoseRateMlph := 40, RequestComplete := ADR(bDoseRequestComplete), RequestAccepted => bDoseRequestSent); // change arbitrary 40 lph to a variable based on dose amount
		ELSIF nPIDPHError < 0 AND bDoseRequestSent = FALSE THEN
			fbDosingPump_phDown.executeDose(DoseQtyMls := LREAL_TO_UINT(nPIDPHOutput), DoseRateMlph := 40, RequestComplete := ADR(bDoseRequestComplete), RequestAccepted => bDoseRequestSent); // change arbitrary 40 lph to a variable based on dose amount
		ELSIF bDoseRequestSent = TRUE AND bDoseRequestComplete = TRUE THEN
			bDoseRequestSent 	:= FALSE;
			bDoseRequestComplete:= FALSE;
		END_IF
		eSMState := WAIT_TRIG;
END_CASE

METHOD FB_init : BOOL
VAR_INPUT
	bInitRetains : BOOL; // if TRUE, the retain variables are initialized (warm start / cold start)
	bInCopyCode : BOOL;  // if TRUE, the instance afterwards gets moved into the copy code (online change)
	
	DosingPump_phUp:  			I_PumpDosing;
	DosingPump_phDOwn:  		I_PumpDosing;

	Sensor_PH:				I_Sensor(SensorID := '', SensorDescr := '' , SensorType := E_SensorType.Analogue);
	Sensor_TEMP:			I_Sensor(SensorID := '', SensorDescr := '' , SensorType := E_SensorType.Analogue);
	
END_VAR
fbDosingPump_phUp := DosingPump_phUp;
fbDosingPump_phDOwn := DosingPump_phDOwn;

fbSensor_PH := Sensor_PH;
fbSensor_TEMP := Sensor_TEMP;
END_METHOD

METHOD initPIDLoops : BOOL
VAR_INPUT
END_VAR
stPIDPHParameters.tCtrlCycleTime := tPIDPHCtrlCycleTime;
stPIDPHParameters.tTaskCycleTime := tPIDPHTaskCycleTime;
stPIDPHParameters.fKp := nPIDPHKp;
stPIDPHParameters.tTn := tPIDPHTn;
stPIDPHParameters.tTv := tPIDPHTv;
stPIDPHParameters.tTd := tPIDPHTd;
stPIDPHParameters.fOutMaxLimit := nPIDPHOutMaxLimit;
stPIDPHParameters.fOutMinLimit := nPIDPHOutMinLimit;
stPIDPHParameters.bPInTheFeedbackPath := bPIDPHPInTheFeedbackPath;
stPIDPHParameters.bDInTheFeedbackPath := bPIDPHDInTheFeedbackPath;
stPIDPHParameters.bARWOnIPartOnly := bPIDPHARWOnIPartOnly;
END_METHOD

METHOD setParams : BOOL
VAR_INPUT
	
	PHMaxDoseRate: UINT;
	PHMinDoseRate: UINT;
	PHTimeBetweenDoses: TIME;
	
	PHSetpoint:				REAL; 
	PHSetpointBand:			REAL;
	PHManSyncVal:			REAL;
	PHSync: 				BOOL;
	PHHold: 				BOOL;
	PHMode: 				E_CTRL_MODE;
	PHCtrlCycleTime: 		TIME;
	PHTaskCycleTime:		TIME;
	
	
	//stPIDParams values
	PHKp:  					REAL;
	PHTn: 					TIME;
	PHTv:					TIME;
	PHTd:					TIME; 
	PHOutMaxLimit: 			REAL; 		
	PHOutMinLimit:			REAL;
	PHPInTheFeedbackPath: 	BOOL;
	PHDInTheFeedbackPath:	BOOL;
	PHARWOnIPartOnly:		BOOL;

END_VAR

nPIDPHMaxDoseRate := PHMaxDoseRate;
nPIDPHMinDoseRate := PHMinDoseRate;
tPIDPHTimeBetweenDoses := PHTimeBetweenDoses;


nPIDPHSetpoint := PHSetpoint;
nPIDPHSetpointBand := PHSetpointBand;
nPIDPHManSyncVal := PHManSyncVal;
bPIDPHSync := PHSync;
bPIDPHHold := PHHold;
ePIDPHMode := PHMode;
tPIDPHCtrlCycleTime := PHCtrlCycleTime;
tPIDPHTaskCycleTime := PHTaskCycleTime;

nPIDPHKp := PHKp;
tPIDPHTn := PHTn;
tPIDPHTv := PHTv;
tPIDPHTd := PHTd;
nPIDPHOutMaxLimit := PHOutMaxLimit;
nPIDPHOutMinLimit := PHOutMinLimit;
bPIDPHPInTheFeedbackPath := PHPInTheFeedbackPath;
bPIDPHDInTheFeedbackPath := PHDInTheFeedbackPath;
bPIDPHARWactive := PHARWOnIPartOnly;
END_METHOD

END_FUNCTION_BLOCK

// ---- POUs/04 Control Loops/Dosing Machine/FB_ControlLoop_PID.TcPOU
FUNCTION_BLOCK FB_ControlLoop_PID EXTENDS FB_BaseDevice


